LIN {X 0,Y 532.059,Z 786.23,A -85,B 0,C 180,E1 -4333.229,E2 -4333.229} C_VEL
LIN {X 0,Y 530.415,Z 776.665,A -85,B 0,C 180,E1 -4333.53,E2 -4333.53} C_VEL
LIN {X 0,Y 530.416,Z 773.451,A -85,B 0,C 180,E1 -4336.156,E2 -4336.156} C_VEL
LIN {X 0,Y 530.403,Z 770.567,A -85,B 0,C 180,E1 -4338.543,E2 -4338.543} C_VEL
LIN {X 0,Y 530.453,Z 767.793,A -85,B 0,C 180,E1 -4340.961,E2 -4340.961} C_VEL
LIN {X 0,Y 530.507,Z 764.565,A -85,B 0,C 180,E1 -4343.922,E2 -4343.922} C_VEL
LIN {X 0,Y 530.506,Z 761.259,A -85,B 0,C 180,E1 -4346.771,E2 -4346.771} C_VEL
LIN {X 0,Y 530.49,Z 757.968,A -85,B 0,C 180,E1 -4349.353,E2 -4349.353} C_VEL
LIN {X 0,Y 530.48,Z 755.565,A -85,B 0,C 180,E1 -4351.111,E2 -4351.111} C_VEL
LIN {X 0,Y 530.791,Z 755.371,A -85,B 0,C 180,E1 -4353.788,E2 -4353.788} C_VEL
LIN {X 0,Y 530.947,Z 755.346,A -85,B 0,C 180,E1 -4356.56,E2 -4356.56} C_VEL
LIN {X 0,Y 530.992,Z 755.343,A -85,B 0,C 180,E1 -4359.444,E2 -4359.444} C_VEL
LIN {X 0,Y 530.968,Z 755.343,A -85,B 0,C 180,E1 -4362.458,E2 -4362.458} C_VEL
LIN {X 0,Y 530.99,Z 755.342,A -85,B 0,C 180,E1 -4365.453,E2 -4365.453} C_VEL
LIN {X 0,Y 530.998,Z 755.342,A -85,B 0,C 180,E1 -4368.565,E2 -4368.565} C_VEL
LIN {X 0,Y 530.992,Z 755.408,A -85,B 0,C 180,E1 -4371.744,E2 -4371.744} C_VEL
LIN {X 0,Y 532.042,Z 761.565,A -85,B 0,C 180,E1 -4374.093,E2 -4374.093} C_VEL
LIN {X 0,Y 532.013,Z 767.898,A -85,B 0,C 180,E1 -4376.33,E2 -4376.33} C_VEL
LIN {X 0,Y 531.734,Z 776.441,A -85,B 0,C 180,E1 -4379.218,E2 -4379.218} C_VEL
LIN {X 0,Y 531.516,Z 785.016,A -85,B 0,C 180,E1 -4382.005,E2 -4382.005} C_VEL
LIN {X 0,Y 531.294,Z 794.397,A -85,B 0,C 180,E1 -4384.957,E2 -4384.957} C_VEL
LIN {X 0,Y 531.163,Z 803.886,A -85,B 0,C 180,E1 -4387.85,E2 -4387.85} C_VEL
LIN {X 0,Y 530.969,Z 813.168,A -85,B 0,C 180,E1 -4390.676,E2 -4390.676} C_VEL
LIN {X 0,Y 530.828,Z 822.435,A -85,B 0,C 180,E1 -4393.462,E2 -4393.462} C_VEL
LIN {X 0,Y 530.706,Z 832.53,A -85,B 0,C 180,E1 -4396.454,E2 -4396.454} C_VEL
LIN {X 0,Y 532.33,Z 843.349,A -85,B 0,C 180,E1 -4396.739,E2 -4396.739} C_VEL
LIN {X 0,Y 532.127,Z 856.77,A -85,B 0,C 180,E1 -4397.171,E2 -4397.171} C_VEL
LIN {X 0,Y 531.869,Z 868.408,A -85,B 0,C 180,E1 -4397.697,E2 -4397.697} C_VEL
LIN {X 0,Y 531.655,Z 879.403,A -85,B 0,C 180,E1 -4398.347,E2 -4398.347} C_VEL
LIN {X 0,Y 531.411,Z 890.095,A -85,B 0,C 180,E1 -4399.137,E2 -4399.137} C_VEL
LIN {X 0,Y 531.128,Z 900.539,A -85,B 0,C 180,E1 -4400.095,E2 -4400.095} C_VEL
LIN {X 0,Y 530.931,Z 908.991,A -85,B 0,C 180,E1 -4401.052,E2 -4401.052} C_VEL
LIN {X 0,Y 530.759,Z 917.236,A -85,B 0,C 180,E1 -4402.199,E2 -4402.199} C_VEL
LIN {X 0,Y 530.599,Z 924.271,A -85,B 0,C 180,E1 -4403.42,E2 -4403.42} C_VEL
LIN {X 0,Y 530.525,Z 929.95,A -85,B 0,C 180,E1 -4404.679,E2 -4404.679} C_VEL
LIN {X 0,Y 530.523,Z 933.895,A -85,B 0,C 180,E1 -4405.822,E2 -4405.822} C_VEL
LIN {X 0,Y 530.457,Z 936.807,A -85,B 0,C 180,E1 -4406.962,E2 -4406.962} C_VEL
LIN {X 0,Y 530.41,Z 938.196,A -85,B 0,C 180,E1 -4407.722,E2 -4407.722} C_VEL
LIN {X 0,Y 530.344,Z 939.786,A -85,B 0,C 180,E1 -4409.241,E2 -4409.241} C_VEL
LIN {X 0,Y 530.343,Z 940,A -85,B 0,C 180,E1 -4410,E2 -4410} C_VEL
LIN {X 0,Y 530.361,Z 939.185,A -85,B 0,C 180,E1 -4411.519,E2 -4411.519} C_VEL
LIN {X 0,Y 530.41,Z 938.198,A -85,B 0,C 180,E1 -4412.278,E2 -4412.278} C_VEL
LIN {X 0,Y 530.457,Z 936.81,A -85,B 0,C 180,E1 -4413.038,E2 -4413.038} C_VEL
LIN {X 0,Y 530.523,Z 933.895,A -85,B 0,C 180,E1 -4414.178,E2 -4414.178} C_VEL
LIN {X 0,Y 530.525,Z 929.948,A -85,B 0,C 180,E1 -4415.321,E2 -4415.321} C_VEL
LIN {X 0,Y 530.599,Z 924.268,A -85,B 0,C 180,E1 -4416.581,E2 -4416.581} C_VEL
LIN {X 0,Y 530.759,Z 917.236,A -85,B 0,C 180,E1 -4417.801,E2 -4417.801} C_VEL
LIN {X 0,Y 530.931,Z 908.991,A -85,B 0,C 180,E1 -4418.948,E2 -4418.948} C_VEL
LIN {X 0,Y 531.112,Z 900.539,A -85,B 0,C 180,E1 -4419.906,E2 -4419.906} C_VEL
LIN {X 0,Y 531.411,Z 890.094,A -85,B 0,C 180,E1 -4420.863,E2 -4420.863} C_VEL
LIN {X 0,Y 531.696,Z 878.247,A -85,B 0,C 180,E1 -4421.731,E2 -4421.731} C_VEL
LIN {X 0,Y 531.921,Z 866.488,A -85,B 0,C 180,E1 -4422.398,E2 -4422.398} C_VEL
LIN {X 0,Y 532.161,Z 854.165,A -85,B 0,C 180,E1 -4422.926,E2 -4422.926} C_VEL
LIN {X 0,Y 532.183,Z 841.514,A -85,B 0,C 180,E1 -4423.314,E2 -4423.314} C_VEL
LIN {X 0,Y 530.706,Z 832.53,A -85,B 0,C 180,E1 -4423.546,E2 -4423.546} C_VEL
LIN {X 0,Y 530.828,Z 822.435,A -85,B 0,C 180,E1 -4426.538,E2 -4426.538} C_VEL
LIN {X 0,Y 530.968,Z 813.168,A -85,B 0,C 180,E1 -4429.324,E2 -4429.324} C_VEL
LIN {X 0,Y 531.163,Z 803.882,A -85,B 0,C 180,E1 -4432.15,E2 -4432.15} C_VEL
LIN {X 0,Y 531.268,Z 794.03,A -85,B 0,C 180,E1 -4435.044,E2 -4435.044} C_VEL
LIN {X 0,Y 531.414,Z 784.276,A -85,B 0,C 180,E1 -4438.001,E2 -4438.001} C_VEL
LIN {X 0,Y 531.62,Z 774.782,A -85,B 0,C 180,E1 -4441.036,E2 -4441.036} C_VEL
LIN {X 0,Y 531.858,Z 767.114,A -85,B 0,C 180,E1 -4443.71,E2 -4443.71} C_VEL
LIN {X 0,Y 532.032,Z 762.369,A -85,B 0,C 180,E1 -4445.537,E2 -4445.537} C_VEL
LIN {X 0,Y 531.466,Z 758.043,A -85,B 0,C 180,E1 -4447.492,E2 -4447.492} C_VEL
LIN {X 0,Y 530.983,Z 755.347,A -85,B 0,C 180,E1 -4449.015,E2 -4449.015} C_VEL
LIN {X 0,Y 530.987,Z 755.344,A -85,B 0,C 180,E1 -4452.166,E2 -4452.166} C_VEL
LIN {X 0,Y 530.989,Z 755.345,A -85,B 0,C 180,E1 -4455.453,E2 -4455.453} C_VEL
LIN {X 0,Y 530.983,Z 755.345,A -85,B 0,C 180,E1 -4458.563,E2 -4458.563} C_VEL
LIN {X 0,Y 530.959,Z 755.347,A -85,B 0,C 180,E1 -4461.529,E2 -4461.529} C_VEL
LIN {X 0,Y 530.929,Z 755.353,A -85,B 0,C 180,E1 -4464.377,E2 -4464.377} C_VEL
LIN {X 0,Y 530.909,Z 755.357,A -85,B 0,C 180,E1 -4465.304,E2 -4465.304} C_VEL
LIN {X 0,Y 530.826,Z 756.592,A -85,B 0,C 180,E1 -4467.123,E2 -4467.123} C_VEL
LIN {X 0,Y 530.714,Z 759.006,A -85,B 0,C 180,E1 -4469.786,E2 -4469.786} C_VEL
LIN {X 0,Y 530.622,Z 761.58,A -85,B 0,C 180,E1 -4472.549,E2 -4472.549} C_VEL
LIN {X 0,Y 530.564,Z 763.83,A -85,B 0,C 180,E1 -4474.92,E2 -4474.92} C_VEL
LIN {X 0,Y 530.51,Z 766.833,A -85,B 0,C 180,E1 -4478.024,E2 -4478.024} C_VEL
LIN {X 0,Y 530.425,Z 769.498,A -85,B 0,C 180,E1 -4480.655,E2 -4480.655} C_VEL
LIN {X 0,Y 530.429,Z 772.38,A -85,B 0,C 180,E1 -4483.052,E2 -4483.052} C_VEL
LIN {X 0,Y 530.43,Z 776.224,A -85,B 0,C 180,E1 -4486.202,E2 -4486.202} C_VEL
LIN {X 0,Y 530.44,Z 776.674,A -85,B 0,C 180,E1 -4486.568,E2 -4486.568} C_VEL
LIN {X 0,Y 532.261,Z 788.537,A -85,B 0,C 180,E1 -4486.931,E2 -4486.931} C_VEL
LIN {X 0,Y 532.013,Z 801.428,A -85,B 0,C 180,E1 -4487.41,E2 -4487.41} C_VEL
LIN {X 0,Y 531.83,Z 813.17,A -85,B 0,C 180,E1 -4488.005,E2 -4488.005} C_VEL
LIN {X 0,Y 531.551,Z 824.586,A -85,B 0,C 180,E1 -4488.753,E2 -4488.753} C_VEL
LIN {X 0,Y 531.282,Z 835.099,A -85,B 0,C 180,E1 -4489.616,E2 -4489.616} C_VEL
LIN {X 0,Y 531.071,Z 843.691,A -85,B 0,C 180,E1 -4490.478,E2 -4490.478} C_VEL
LIN {X 0,Y 530.892,Z 851.608,A -85,B 0,C 180,E1 -4491.434,E2 -4491.434} C_VEL
LIN {X 0,Y 530.69,Z 859.354,A -85,B 0,C 180,E1 -4492.58,E2 -4492.58} C_VEL
LIN {X 0,Y 530.603,Z 866.462,A -85,B 0,C 180,E1 -4493.917,E2 -4493.917} C_VEL
LIN {X 0,Y 530.46,Z 871.201,A -85,B 0,C 180,E1 -4495.059,E2 -4495.059} C_VEL
LIN {X 0,Y 530.516,Z 874.833,A -85,B 0,C 180,E1 -4496.201,E2 -4496.201} C_VEL
LIN {X 0,Y 530.458,Z 876.708,A -85,B 0,C 180,E1 -4496.961,E2 -4496.961} C_VEL
LIN {X 0,Y 530.411,Z 878.13,A -85,B 0,C 180,E1 -4497.721,E2 -4497.721} C_VEL
LIN {X 0,Y 530.345,Z 879.758,A -85,B 0,C 180,E1 -4499.24,E2 -4499.24} C_VEL
LIN {X 0,Y 530.343,Z 879.996,A -85,B 0,C 180,E1 -4499.999,E2 -4499.999} C_VEL
LIN {X 0,Y 530.344,Z 879.814,A -85,B 0,C 180,E1 -4500.759,E2 -4500.759} C_VEL
LIN {X 0,Y 530.41,Z 878.263,A -85,B 0,C 180,E1 -4502.277,E2 -4502.277} C_VEL
LIN {X 0,Y 530.457,Z 876.902,A -85,B 0,C 180,E1 -4503.037,E2 -4503.037} C_VEL
LIN {X 0,Y 530.523,Z 874.023,A -85,B 0,C 180,E1 -4504.177,E2 -4504.177} C_VEL
LIN {X 0,Y 530.523,Z 870.121,A -85,B 0,C 180,E1 -4505.32,E2 -4505.32} C_VEL
LIN {X 0,Y 530.592,Z 864.537,A -85,B 0,C 180,E1 -4506.575,E2 -4506.575} C_VEL
LIN {X 0,Y 530.757,Z 857.531,A -85,B 0,C 180,E1 -4507.8,E2 -4507.8} C_VEL
LIN {X 0,Y 530.927,Z 849.347,A -85,B 0,C 180,E1 -4508.947,E2 -4508.947} C_VEL
LIN {X 0,Y 531.106,Z 840.977,A -85,B 0,C 180,E1 -4509.905,E2 -4509.905} C_VEL
LIN {X 0,Y 531.404,Z 830.653,A -85,B 0,C 180,E1 -4510.862,E2 -4510.862} C_VEL
LIN {X 0,Y 531.643,Z 818.958,A -85,B 0,C 180,E1 -4511.729,E2 -4511.729} C_VEL
LIN {X 0,Y 531.868,Z 807.425,A -85,B 0,C 180,E1 -4512.398,E2 -4512.398} C_VEL
LIN {X 0,Y 532.131,Z 795.405,A -85,B 0,C 180,E1 -4512.925,E2 -4512.925} C_VEL
LIN {X 0,Y 532.125,Z 786.435,A -85,B 0,C 180,E1 -4513.229,E2 -4513.229} C_VEL
LIN {X 0,Y 530.414,Z 776.667,A -85,B 0,C 180,E1 -4513.529,E2 -4513.529} C_VEL
LIN {X 0,Y 530.411,Z 773.452,A -85,B 0,C 180,E1 -4516.155,E2 -4516.155} C_VEL
LIN {X 0,Y 530.399,Z 770.569,A -85,B 0,C 180,E1 -4518.542,E2 -4518.542} C_VEL
LIN {X 0,Y 530.441,Z 767.695,A -85,B 0,C 180,E1 -4520.96,E2 -4520.96} C_VEL
LIN {X 0,Y 530.514,Z 764.314,A -85,B 0,C 180,E1 -4523.924,E2 -4523.924} C_VEL
LIN {X 0,Y 530.526,Z 761.426,A -85,B 0,C 180,E1 -4526.769,E2 -4526.769} C_VEL
LIN {X 0,Y 530.558,Z 758.697,A -85,B 0,C 180,E1 -4529.347,E2 -4529.347} C_VEL
LIN {X 0,Y 530.622,Z 755.781,A -85,B 0,C 180,E1 -4532.04,E2 -4532.04} C_VEL
LIN {X 0,Y 530.783,Z 755.372,A -85,B 0,C 180,E1 -4533.786,E2 -4533.786} C_VEL
LIN {X 0,Y 530.941,Z 755.345,A -85,B 0,C 180,E1 -4536.558,E2 -4536.558} C_VEL
LIN {X 0,Y 530.975,Z 755.344,A -85,B 0,C 180,E1 -4539.57,E2 -4539.57} C_VEL
LIN {X 0,Y 530.3,Z 755.427,A -85,B 0,C 180,E1 -4540.203,E2 -4540.203} C_VEL
LIN {X 0,Y 527.438,Z 755.788,A -85,B 0,C 180,E1 -4541.23,E2 -4541.23} C_VEL
LIN {X 0,Y 525.026,Z 756.084,A -85,B 0,C 180,E1 -4542.057,E2 -4542.057} C_VEL
LIN {X 0,Y 523.992,Z 756.212,A -85,B 0,C 180,E1 -4542.696,E2 -4542.696} C_VEL
LIN {X 0,Y 523.909,Z 756.224,A -85,B 0,C 180,E1 -4542.912,E2 -4542.912} C_VEL
LIN {X 0,Y 523.936,Z 756.221,A -85,B 0,C 180,E1 -4545.771,E2 -4545.771} C_VEL
LIN {X 0,Y 523.932,Z 756.22,A -85,B 0,C 180,E1 -4548.907,E2 -4548.907} C_VEL
LIN {X 0,Y 523.908,Z 756.223,A -85,B 0,C 180,E1 -4551.897,E2 -4551.897} C_VEL
LIN {X 0,Y 523.916,Z 756.221,A -85,B 0,C 180,E1 -4554.911,E2 -4554.911} C_VEL
LIN {X 0,Y 523.927,Z 756.224,A -85,B 0,C 180,E1 -4557.679,E2 -4557.679} C_VEL
LIN {X 0,Y 523.945,Z 756.216,A -85,B 0,C 180,E1 -4560.676,E2 -4560.676} C_VEL
LIN {X 0,Y 523.925,Z 756.225,A -85,B 0,C 180,E1 -4563.726,E2 -4563.726} C_VEL
LIN {X 0,Y 523.9,Z 756.223,A -85,B 0,C 180,E1 -4566.269,E2 -4566.269} C_VEL
LIN {X 0,Y 523.936,Z 756.216,A -85,B 0,C 180,E1 -4568.766,E2 -4568.766} C_VEL
LIN {X 0,Y 523.928,Z 756.219,A -85,B 0,C 180,E1 -4571.22,E2 -4571.22} C_VEL
LIN {X 0,Y 523.916,Z 756.226,A -85,B 0,C 180,E1 -4573.638,E2 -4573.638} C_VEL
LIN {X 0,Y 523.921,Z 756.224,A -85,B 0,C 180,E1 -4576.027,E2 -4576.027} C_VEL
LIN {X 0,Y 523.979,Z 756.211,A -85,B 0,C 180,E1 -4579.177,E2 -4579.177} C_VEL
LIN {X 0,Y 523.942,Z 756.219,A -85,B 0,C 180,E1 -4581.515,E2 -4581.515} C_VEL
LIN {X 0,Y 524.02,Z 756.206,A -85,B 0,C 180,E1 -4584.613,E2 -4584.613} C_VEL
LIN {X 0,Y 524.093,Z 756.201,A -85,B 0,C 180,E1 -4587.694,E2 -4587.694} C_VEL
LIN {X 0,Y 524.085,Z 756.206,A -85,B 0,C 180,E1 -4590,E2 -4590} C_VEL
LIN {X 0,Y 524.09,Z 756.202,A -85,B 0,C 180,E1 -4592.306,E2 -4592.306} C_VEL
LIN {X 0,Y 523.991,Z 756.218,A -85,B 0,C 180,E1 -4596.16,E2 -4596.16} C_VEL
LIN {X 0,Y 523.933,Z 756.216,A -85,B 0,C 180,E1 -4599.263,E2 -4599.263} C_VEL
LIN {X 0,Y 523.941,Z 756.222,A -85,B 0,C 180,E1 -4602.393,E2 -4602.393} C_VEL
LIN {X 0,Y 523.914,Z 756.219,A -85,B 0,C 180,E1 -4605.563,E2 -4605.563} C_VEL
LIN {X 0,Y 523.906,Z 756.224,A -85,B 0,C 180,E1 -4607.971,E2 -4607.971} C_VEL
LIN {X 0,Y 523.962,Z 756.222,A -85,B 0,C 180,E1 -4610.411,E2 -4610.411} C_VEL
LIN {X 0,Y 523.899,Z 756.223,A -85,B 0,C 180,E1 -4612.894,E2 -4612.894} C_VEL
LIN {X 0,Y 523.89,Z 756.222,A -85,B 0,C 180,E1 -4615.422,E2 -4615.422} C_VEL
LIN {X 0,Y 523.906,Z 756.223,A -85,B 0,C 180,E1 -4618.003,E2 -4618.003} C_VEL
LIN {X 0,Y 523.931,Z 756.222,A -85,B 0,C 180,E1 -4620.854,E2 -4620.854} C_VEL
LIN {X 0,Y 523.922,Z 756.219,A -85,B 0,C 180,E1 -4623.73,E2 -4623.73} C_VEL
LIN {X 0,Y 523.896,Z 756.227,A -85,B 0,C 180,E1 -4626.402,E2 -4626.402} C_VEL
LIN {X 0,Y 523.913,Z 756.223,A -85,B 0,C 180,E1 -4629.086,E2 -4629.086} C_VEL
LIN {X 0,Y 523.945,Z 756.217,A -85,B 0,C 180,E1 -4632.12,E2 -4632.12} C_VEL
LIN {X 0,Y 523.937,Z 756.219,A -85,B 0,C 180,E1 -4635.311,E2 -4635.311} C_VEL
LIN {X 0,Y 523.951,Z 756.221,A -85,B 0,C 180,E1 -4638.691,E2 -4638.691} C_VEL
LIN {X 0,Y 523.912,Z 756.226,A -85,B 0,C 180,E1 -4641.082,E2 -4641.082} C_VEL
LIN {X 0,Y 523.893,Z 756.222,A -85,B 0,C 180,E1 -4643.826,E2 -4643.826} C_VEL
LIN {X 0,Y 523.722,Z 756.251,A -85,B 0,C 180,E1 -4646.621,E2 -4646.621} C_VEL
LIN {X 0,Y 523.505,Z 756.279,A -85,B 0,C 180,E1 -4648.429,E2 -4648.429} C_VEL
LIN {X 0,Y 523.434,Z 759.216,A -85,B 0,C 180,E1 -4651.096,E2 -4651.096} C_VEL
LIN {X 0,Y 523.464,Z 762.594,A -85,B 0,C 180,E1 -4654.098,E2 -4654.098} C_VEL
LIN {X 0,Y 523.385,Z 765.959,A -85,B 0,C 180,E1 -4657.083,E2 -4657.083} C_VEL
LIN {X 0,Y 523.379,Z 769.308,A -85,B 0,C 180,E1 -4660.047,E2 -4660.047} C_VEL
LIN {X 0,Y 523.338,Z 772.383,A -85,B 0,C 180,E1 -4662.817,E2 -4662.817} C_VEL
LIN {X 0,Y 523.364,Z 776.587,A -85,B 0,C 180,E1 -4666.31,E2 -4666.31} C_VEL
LIN {X 0,Y 523.363,Z 776.677,A -85,B 0,C 180,E1 -4666.385,E2 -4666.385} C_VEL
LIN {X 0,Y 525.294,Z 788.698,A -85,B 0,C 180,E1 -4666.756,E2 -4666.756} C_VEL
LIN {X 0,Y 525.059,Z 801.414,A -85,B 0,C 180,E1 -4667.242,E2 -4667.242} C_VEL
LIN {X 0,Y 524.826,Z 811.363,A -85,B 0,C 180,E1 -4667.742,E2 -4667.742} C_VEL
LIN {X 0,Y 524.67,Z 821.852,A -85,B 0,C 180,E1 -4668.41,E2 -4668.41} C_VEL
LIN {X 0,Y 524.401,Z 830.657,A -85,B 0,C 180,E1 -4669.089,E2 -4669.089} C_VEL
LIN {X 0,Y 524.179,Z 838.123,A -85,B 0,C 180,E1 -4669.768,E2 -4669.768} C_VEL
LIN {X 0,Y 523.99,Z 845.395,A -85,B 0,C 180,E1 -4670.544,E2 -4670.544} C_VEL
LIN {X 0,Y 523.794,Z 852.985,A -85,B 0,C 180,E1 -4671.513,E2 -4671.513} C_VEL
LIN {X 0,Y 523.636,Z 859.318,A -85,B 0,C 180,E1 -4672.482,E2 -4672.482} C_VEL
LIN {X 0,Y 523.528,Z 864.446,A -85,B 0,C 180,E1 -4673.415,E2 -4673.415} C_VEL
LIN {X 0,Y 523.464,Z 869.72,A -85,B 0,C 180,E1 -4674.608,E2 -4674.608} C_VEL
LIN {X 0,Y 523.441,Z 873.701,A -85,B 0,C 180,E1 -4675.766,E2 -4675.766} C_VEL
LIN {X 0,Y 523.367,Z 876.652,A -85,B 0,C 180,E1 -4676.922,E2 -4676.922} C_VEL
LIN {X 0,Y 523.334,Z 878.143,A -85,B 0,C 180,E1 -4677.692,E2 -4677.692} C_VEL
LIN {X 0,Y 523.25,Z 879.719,A -85,B 0,C 180,E1 -4679.231,E2 -4679.231} C_VEL
LIN {X 0,Y 523.247,Z 879.999,A -85,B 0,C 180,E1 -4680.001,E2 -4680.001} C_VEL
LIN {X 0,Y 523.275,Z 879.2,A -85,B 0,C 180,E1 -4681.54,E2 -4681.54} C_VEL
LIN {X 0,Y 523.334,Z 878.278,A -85,B 0,C 180,E1 -4682.31,E2 -4682.31} C_VEL
LIN {X 0,Y 523.444,Z 875.036,A -85,B 0,C 180,E1 -4683.85,E2 -4683.85} C_VEL
LIN {X 0,Y 523.383,Z 871.477,A -85,B 0,C 180,E1 -4685.008,E2 -4685.008} C_VEL
LIN {X 0,Y 523.537,Z 868.573,A -85,B 0,C 180,E1 -4685.779,E2 -4685.779} C_VEL
LIN {X 0,Y 523.584,Z 862.019,A -85,B 0,C 180,E1 -4687.133,E2 -4687.133} C_VEL
LIN {X 0,Y 523.723,Z 856.229,A -85,B 0,C 180,E1 -4688.101,E2 -4688.101} C_VEL
LIN {X 0,Y 523.867,Z 849.264,A -85,B 0,C 180,E1 -4689.07,E2 -4689.07} C_VEL
LIN {X 0,Y 524.051,Z 842.707,A -85,B 0,C 180,E1 -4689.846,E2 -4689.846} C_VEL
LIN {X 0,Y 524.285,Z 833.886,A -85,B 0,C 180,E1 -4690.72,E2 -4690.72} C_VEL
LIN {X 0,Y 524.545,Z 825.715,A -85,B 0,C 180,E1 -4691.399,E2 -4691.399} C_VEL
LIN {X 0,Y 524.715,Z 816.442,A -85,B 0,C 180,E1 -4692.043,E2 -4692.043} C_VEL
LIN {X 0,Y 524.97,Z 807.257,A -85,B 0,C 180,E1 -4692.566,E2 -4692.566} C_VEL
LIN {X 0,Y 525.192,Z 796.453,A -85,B 0,C 180,E1 -4693.052,E2 -4693.052} C_VEL
LIN {X 0,Y 525.151,Z 787.293,A -85,B 0,C 180,E1 -4693.376,E2 -4693.376} C_VEL
LIN {X 0,Y 523.353,Z 776.664,A -85,B 0,C 180,E1 -4693.716,E2 -4693.716} C_VEL
LIN {X 0,Y 523.315,Z 773.45,A -85,B 0,C 180,E1 -4696.382,E2 -4696.382} C_VEL
LIN {X 0,Y 523.315,Z 770.726,A -85,B 0,C 180,E1 -4698.804,E2 -4698.804} C_VEL
LIN {X 0,Y 523.384,Z 768.119,A -85,B 0,C 180,E1 -4701.258,E2 -4701.258} C_VEL
LIN {X 0,Y 523.429,Z 765.314,A -85,B 0,C 180,E1 -4703.754,E2 -4703.754} C_VEL
LIN {X 0,Y 523.431,Z 762.363,A -85,B 0,C 180,E1 -4706.301,E2 -4706.301} C_VEL
LIN {X 0,Y 523.417,Z 758.654,A -85,B 0,C 180,E1 -4709.218,E2 -4709.218} C_VEL
LIN {X 0,Y 523.396,Z 756.574,A -85,B 0,C 180,E1 -4710.753,E2 -4710.753} C_VEL
LIN {X 0,Y 523.597,Z 756.267,A -85,B 0,C 180,E1 -4712.474,E2 -4712.474} C_VEL
LIN {X 0,Y 523.865,Z 756.234,A -85,B 0,C 180,E1 -4715.232,E2 -4715.232} C_VEL
LIN {X 0,Y 523.919,Z 756.22,A -85,B 0,C 180,E1 -4718.102,E2 -4718.102} C_VEL
LIN {X 0,Y 523.939,Z 756.224,A -85,B 0,C 180,E1 -4721.093,E2 -4721.093} C_VEL
LIN {X 0,Y 523.939,Z 756.218,A -85,B 0,C 180,E1 -4724.229,E2 -4724.229} C_VEL
LIN {X 0,Y 523.922,Z 756.226,A -85,B 0,C 180,E1 -4726.833,E2 -4726.833} C_VEL
LIN {X 0,Y 523.944,Z 756.224,A -85,B 0,C 180,E1 -4728.908,E2 -4728.908} C_VEL
LIN {X 0,Y 523.949,Z 756.275,A -85,B 0,C 180,E1 -4731.472,E2 -4731.472} C_VEL
LIN {X 0,Y 525.035,Z 762.583,A -85,B 0,C 180,E1 -4733.916,E2 -4733.916} C_VEL
LIN {X 0,Y 525.09,Z 767.758,A -85,B 0,C 180,E1 -4735.796,E2 -4735.796} C_VEL
LIN {X 0,Y 524.805,Z 775.632,A -85,B 0,C 180,E1 -4738.515,E2 -4738.515} C_VEL
LIN {X 0,Y 524.524,Z 784.894,A -85,B 0,C 180,E1 -4741.598,E2 -4741.598} C_VEL
LIN {X 0,Y 524.328,Z 793.131,A -85,B 0,C 180,E1 -4744.249,E2 -4744.249} C_VEL
LIN {X 0,Y 524.129,Z 802.291,A -85,B 0,C 180,E1 -4747.116,E2 -4747.116} C_VEL
LIN {X 0,Y 523.996,Z 811.37,A -85,B 0,C 180,E1 -4749.862,E2 -4749.862} C_VEL
LIN {X 0,Y 523.821,Z 821.111,A -85,B 0,C 180,E1 -4752.832,E2 -4752.832} C_VEL
LIN {X 0,Y 523.659,Z 831.703,A -85,B 0,C 180,E1 -4756.02,E2 -4756.02} C_VEL
LIN {X 0,Y 523.652,Z 832.725,A -85,B 0,C 180,E1 -4756.286,E2 -4756.286} C_VEL
LIN {X 0,Y 525.427,Z 844.264,A -85,B 0,C 180,E1 -4756.586,E2 -4756.586} C_VEL
LIN {X 0,Y 525.216,Z 856.771,A -85,B 0,C 180,E1 -4756.999,E2 -4756.999} C_VEL
LIN {X 0,Y 524.934,Z 868.407,A -85,B 0,C 180,E1 -4757.532,E2 -4757.532} C_VEL
LIN {X 0,Y 524.684,Z 879.822,A -85,B 0,C 180,E1 -4758.218,E2 -4758.218} C_VEL
LIN {X 0,Y 524.395,Z 891.264,A -85,B 0,C 180,E1 -4759.088,E2 -4759.088} C_VEL
LIN {X 0,Y 524.106,Z 900.539,A -85,B 0,C 180,E1 -4759.961,E2 -4759.961} C_VEL
LIN {X 0,Y 523.897,Z 908.991,A -85,B 0,C 180,E1 -4760.931,E2 -4760.931} C_VEL
LIN {X 0,Y 523.689,Z 917.236,A -85,B 0,C 180,E1 -4762.093,E2 -4762.093} C_VEL
LIN {X 0,Y 523.576,Z 922.868,A -85,B 0,C 180,E1 -4763.061,E2 -4763.061} C_VEL
LIN {X 0,Y 523.544,Z 928.366,A -85,B 0,C 180,E1 -4764.222,E2 -4764.222} C_VEL
LIN {X 0,Y 523.361,Z 932.677,A -85,B 0,C 180,E1 -4765.379,E2 -4765.379} C_VEL
LIN {X 0,Y 523.444,Z 934.958,A -85,B 0,C 180,E1 -4766.151,E2 -4766.151} C_VEL
LIN {X 0,Y 523.368,Z 936.807,A -85,B 0,C 180,E1 -4766.921,E2 -4766.921} C_VEL
LIN {X 0,Y 523.334,Z 938.195,A -85,B 0,C 180,E1 -4767.691,E2 -4767.691} C_VEL
LIN {X 0,Y 523.25,Z 939.786,A -85,B 0,C 180,E1 -4769.23,E2 -4769.23} C_VEL
LIN {X 0,Y 523.246,Z 940,A -85,B 0,C 180,E1 -4770,E2 -4770} C_VEL
LIN {X 0,Y 523.275,Z 939.185,A -85,B 0,C 180,E1 -4771.539,E2 -4771.539} C_VEL
LIN {X 0,Y 523.334,Z 938.197,A -85,B 0,C 180,E1 -4772.309,E2 -4772.309} C_VEL
LIN {X 0,Y 523.368,Z 936.81,A -85,B 0,C 180,E1 -4773.079,E2 -4773.079} C_VEL
LIN {X 0,Y 523.442,Z 933.895,A -85,B 0,C 180,E1 -4774.235,E2 -4774.235} C_VEL
LIN {X 0,Y 523.464,Z 929.948,A -85,B 0,C 180,E1 -4775.393,E2 -4775.393} C_VEL
LIN {X 0,Y 523.524,Z 924.731,A -85,B 0,C 180,E1 -4776.58,E2 -4776.58} C_VEL
LIN {X 0,Y 523.666,Z 918.467,A -85,B 0,C 180,E1 -4777.713,E2 -4777.713} C_VEL
LIN {X 0,Y 523.857,Z 910.477,A -85,B 0,C 180,E1 -4778.875,E2 -4778.875} C_VEL
LIN {X 0,Y 524.085,Z 902.333,A -85,B 0,C 180,E1 -4779.845,E2 -4779.845} C_VEL
LIN {X 0,Y 524.365,Z 892.398,A -85,B 0,C 180,E1 -4780.815,E2 -4780.815} C_VEL
LIN {X 0,Y 524.666,Z 881.218,A -85,B 0,C 180,E1 -4781.686,E2 -4781.686} C_VEL
LIN {X 0,Y 524.901,Z 870.172,A -85,B 0,C 180,E1 -4782.37,E2 -4782.37} C_VEL
LIN {X 0,Y 525.171,Z 857.973,A -85,B 0,C 180,E1 -4782.953,E2 -4782.953} C_VEL
LIN {X 0,Y 525.387,Z 845.172,A -85,B 0,C 180,E1 -4783.391,E2 -4783.391} C_VEL
LIN {X 0,Y 524.969,Z 840.5,A -85,B 0,C 180,E1 -4783.525,E2 -4783.525} C_VEL
LIN {X 0,Y 523.641,Z 832.53,A -85,B 0,C 180,E1 -4783.733,E2 -4783.733} C_VEL
LIN {X 0,Y 523.796,Z 822.435,A -85,B 0,C 180,E1 -4786.767,E2 -4786.767} C_VEL
LIN {X 0,Y 523.96,Z 813.168,A -85,B 0,C 180,E1 -4789.593,E2 -4789.593} C_VEL
LIN {X 0,Y 524.124,Z 803.086,A -85,B 0,C 180,E1 -4792.545,E2 -4792.545} C_VEL
LIN {X 0,Y 524.252,Z 792.491,A -85,B 0,C 180,E1 -4795.745,E2 -4795.745} C_VEL
LIN {X 0,Y 524.394,Z 783.918,A -85,B 0,C 180,E1 -4798.41,E2 -4798.41} C_VEL
LIN {X 0,Y 524.649,Z 774.575,A -85,B 0,C 180,E1 -4801.495,E2 -4801.495} C_VEL
LIN {X 0,Y 524.95,Z 767.089,A -85,B 0,C 180,E1 -4804.215,E2 -4804.215} C_VEL
LIN {X 0,Y 524.989,Z 762.525,A -85,B 0,C 180,E1 -4806.088,E2 -4806.088} C_VEL
LIN {X 0,Y 524.324,Z 758.472,A -85,B 0,C 180,E1 -4808.067,E2 -4808.067} C_VEL
LIN {X 0,Y 523.958,Z 756.222,A -85,B 0,C 180,E1 -4809.454,E2 -4809.454} C_VEL
LIN {X 0,Y 523.94,Z 756.223,A -85,B 0,C 180,E1 -4812.459,E2 -4812.459} C_VEL
LIN {X 0,Y 523.958,Z 756.222,A -85,B 0,C 180,E1 -4815.309,E2 -4815.309} C_VEL
LIN {X 0,Y 523.944,Z 756.224,A -85,B 0,C 180,E1 -4818.692,E2 -4818.692} C_VEL
LIN {X 0,Y 523.918,Z 756.223,A -85,B 0,C 180,E1 -4821.898,E2 -4821.898} C_VEL
LIN {X 0,Y 523.866,Z 756.234,A -85,B 0,C 180,E1 -4824.921,E2 -4824.921} C_VEL
LIN {X 0,Y 523.805,Z 756.314,A -85,B 0,C 180,E1 -4825.7,E2 -4825.7} C_VEL
LIN {X 0,Y 523.715,Z 758.673,A -85,B 0,C 180,E1 -4828.441,E2 -4828.441} C_VEL
LIN {X 0,Y 523.63,Z 761.076,A -85,B 0,C 180,E1 -4831.106,E2 -4831.106} C_VEL
LIN {X 0,Y 523.531,Z 763.833,A -85,B 0,C 180,E1 -4834.083,E2 -4834.083} C_VEL
LIN {X 0,Y 523.449,Z 766.738,A -85,B 0,C 180,E1 -4837.084,E2 -4837.084} C_VEL
LIN {X 0,Y 523.384,Z 769.554,A -85,B 0,C 180,E1 -4840.046,E2 -4840.046} C_VEL
LIN {X 0,Y 523.342,Z 772.381,A -85,B 0,C 180,E1 -4842.815,E2 -4842.815} C_VEL
LIN {X 0,Y 523.341,Z 776.465,A -85,B 0,C 180,E1 -4846.209,E2 -4846.209} C_VEL
LIN {X 0,Y 523.344,Z 776.675,A -85,B 0,C 180,E1 -4846.382,E2 -4846.382} C_VEL
LIN {X 0,Y 525.347,Z 789.317,A -85,B 0,C 180,E1 -4846.78,E2 -4846.78} C_VEL
LIN {X 0,Y 525.09,Z 801.442,A -85,B 0,C 180,E1 -4847.241,E2 -4847.241} C_VEL
LIN {X 0,Y 524.888,Z 812.537,A -85,B 0,C 180,E1 -4847.806,E2 -4847.806} C_VEL
LIN {X 0,Y 524.585,Z 824.593,A -85,B 0,C 180,E1 -4848.602,E2 -4848.602} C_VEL
LIN {X 0,Y 524.284,Z 835.105,A -85,B 0,C 180,E1 -4849.476,E2 -4849.476} C_VEL
LIN {X 0,Y 524.061,Z 843.697,A -85,B 0,C 180,E1 -4850.349,E2 -4850.349} C_VEL
LIN {X 0,Y 523.86,Z 851.613,A -85,B 0,C 180,E1 -4851.319,E2 -4851.319} C_VEL
LIN {X 0,Y 523.637,Z 859.358,A -85,B 0,C 180,E1 -4852.48,E2 -4852.48} C_VEL
LIN {X 0,Y 523.517,Z 866.465,A -85,B 0,C 180,E1 -4853.834,E2 -4853.834} C_VEL
LIN {X 0,Y 523.384,Z 871.203,A -85,B 0,C 180,E1 -4854.992,E2 -4854.992} C_VEL
LIN {X 0,Y 523.444,Z 874.834,A -85,B 0,C 180,E1 -4856.15,E2 -4856.15} C_VEL
LIN {X 0,Y 523.368,Z 876.71,A -85,B 0,C 180,E1 -4856.92,E2 -4856.92} C_VEL
LIN {X 0,Y 523.335,Z 878.13,A -85,B 0,C 180,E1 -4857.69,E2 -4857.69} C_VEL
LIN {X 0,Y 523.251,Z 879.758,A -85,B 0,C 180,E1 -4859.23,E2 -4859.23} C_VEL
LIN {X 0,Y 523.247,Z 879.997,A -85,B 0,C 180,E1 -4859.999,E2 -4859.999} C_VEL
LIN {X 0,Y 523.25,Z 879.814,A -85,B 0,C 180,E1 -4860.769,E2 -4860.769} C_VEL
LIN {X 0,Y 523.334,Z 878.262,A -85,B 0,C 180,E1 -4862.308,E2 -4862.308} C_VEL
LIN {X 0,Y 523.368,Z 876.9,A -85,B 0,C 180,E1 -4863.078,E2 -4863.078} C_VEL
LIN {X 0,Y 523.441,Z 874.021,A -85,B 0,C 180,E1 -4864.234,E2 -4864.234} C_VEL
LIN {X 0,Y 523.462,Z 870.118,A -85,B 0,C 180,E1 -4865.392,E2 -4865.392} C_VEL
LIN {X 0,Y 523.532,Z 864.375,A -85,B 0,C 180,E1 -4866.691,E2 -4866.691} C_VEL
LIN {X 0,Y 523.687,Z 857.526,A -85,B 0,C 180,E1 -4867.906,E2 -4867.906} C_VEL
LIN {X 0,Y 523.897,Z 849.342,A -85,B 0,C 180,E1 -4869.068,E2 -4869.068} C_VEL
LIN {X 0,Y 524.088,Z 840.971,A -85,B 0,C 180,E1 -4870.039,E2 -4870.039} C_VEL
LIN {X 0,Y 524.418,Z 830.644,A -85,B 0,C 180,E1 -4871.009,E2 -4871.009} C_VEL
LIN {X 0,Y 524.693,Z 820.524,A -85,B 0,C 180,E1 -4871.778,E2 -4871.778} C_VEL
LIN {X 0,Y 524.909,Z 809.232,A -85,B 0,C 180,E1 -4872.467,E2 -4872.467} C_VEL
LIN {X 0,Y 525.167,Z 797.907,A -85,B 0,C 180,E1 -4873.001,E2 -4873.001} C_VEL
LIN {X 0,Y 525.148,Z 787.208,A -85,B 0,C 180,E1 -4873.383,E2 -4873.383} C_VEL
LIN {X 0,Y 523.351,Z 776.666,A -85,B 0,C 180,E1 -4873.715,E2 -4873.715} C_VEL
LIN {X 0,Y 523.311,Z 773.452,A -85,B 0,C 180,E1 -4876.38,E2 -4876.38} C_VEL
LIN {X 0,Y 523.337,Z 769.635,A -85,B 0,C 180,E1 -4879.616,E2 -4879.616} C_VEL
LIN {X 0,Y 523.404,Z 766.858,A -85,B 0,C 180,E1 -4882.104,E2 -4882.104} C_VEL
LIN {X 0,Y 523.424,Z 764.306,A -85,B 0,C 180,E1 -4884.596,E2 -4884.596} C_VEL
LIN {X 0,Y 523.475,Z 761.679,A -85,B 0,C 180,E1 -4887.159,E2 -4887.159} C_VEL
LIN {X 0,Y 523.497,Z 758.794,A -85,B 0,C 180,E1 -4889.783,E2 -4889.783} C_VEL
LIN {X 0,Y 523.552,Z 756.273,A -85,B 0,C 180,E1 -4892.253,E2 -4892.253} C_VEL
LIN {X 0,Y 523.855,Z 756.235,A -85,B 0,C 180,E1 -4895.078,E2 -4895.078} C_VEL
LIN {X 0,Y 523.91,Z 756.22,A -85,B 0,C 180,E1 -4898.101,E2 -4898.101} C_VEL
LIN {X 0,Y 523.935,Z 756.224,A -85,B 0,C 180,E1 -4901.091,E2 -4901.091} C_VEL
LIN {X 0,Y 523.909,Z 756.224,A -85,B 0,C 180,E1 -4902.912,E2 -4902.912} C_VEL
LIN {X 0,Y 523.25,Z 756.311,A -85,B 0,C 180,E1 -4903.554,E2 -4903.554} C_VEL
LIN {X 0,Y 520.411,Z 756.664,A -85,B 0,C 180,E1 -4904.597,E2 -4904.597} C_VEL
LIN {X 0,Y 518.001,Z 756.962,A -85,B 0,C 180,E1 -4905.436,E2 -4905.436} C_VEL
LIN {X 0,Y 516.955,Z 757.088,A -85,B 0,C 180,E1 -4906.085,E2 -4906.085} C_VEL
LIN {X 0,Y 516.864,Z 757.098,A -85,B 0,C 180,E1 -4906.304,E2 -4906.304} C_VEL
LIN {X 0,Y 516.876,Z 757.104,A -85,B 0,C 180,E1 -4909.257,E2 -4909.257} C_VEL
LIN {X 0,Y 516.856,Z 757.099,A -85,B 0,C 180,E1 -4912.273,E2 -4912.273} C_VEL
LIN {X 0,Y 516.871,Z 757.101,A -85,B 0,C 180,E1 -4915.174,E2 -4915.174} C_VEL
LIN {X 0,Y 516.865,Z 757.101,A -85,B 0,C 180,E1 -4917.974,E2 -4917.974} C_VEL
LIN {X 0,Y 516.912,Z 757.092,A -85,B 0,C 180,E1 -4920.695,E2 -4920.695} C_VEL
LIN {X 0,Y 516.891,Z 757.1,A -85,B 0,C 180,E1 -4923.813,E2 -4923.813} C_VEL
LIN {X 0,Y 516.849,Z 757.099,A -85,B 0,C 180,E1 -4926.775,E2 -4926.775} C_VEL
LIN {X 0,Y 516.93,Z 757.097,A -85,B 0,C 180,E1 -4929.731,E2 -4929.731} C_VEL
LIN {X 0,Y 516.887,Z 757.095,A -85,B 0,C 180,E1 -4932.595,E2 -4932.595} C_VEL
LIN {X 0,Y 516.932,Z 757.089,A -85,B 0,C 180,E1 -4935.03,E2 -4935.03} C_VEL
LIN {X 0,Y 516.956,Z 757.089,A -85,B 0,C 180,E1 -4938.233,E2 -4938.233} C_VEL
LIN {X 0,Y 516.919,Z 757.092,A -85,B 0,C 180,E1 -4941.399,E2 -4941.399} C_VEL
LIN {X 0,Y 516.971,Z 757.085,A -85,B 0,C 180,E1 -4944.539,E2 -4944.539} C_VEL
LIN {X 0,Y 517.062,Z 757.076,A -85,B 0,C 180,E1 -4947.663,E2 -4947.663} C_VEL
LIN {X 0,Y 517.054,Z 757.082,A -85,B 0,C 180,E1 -4950,E2 -4950} C_VEL
LIN {X 0,Y 517.06,Z 757.078,A -85,B 0,C 180,E1 -4952.337,E2 -4952.337} C_VEL
LIN {X 0,Y 516.958,Z 757.093,A -85,B 0,C 180,E1 -4956.244,E2 -4956.244} C_VEL
LIN {X 0,Y 516.895,Z 757.093,A -85,B 0,C 180,E1 -4959.39,E2 -4959.39} C_VEL
LIN {X 0,Y 516.894,Z 757.098,A -85,B 0,C 180,E1 -4962.565,E2 -4962.565} C_VEL
LIN {X 0,Y 516.935,Z 757.088,A -85,B 0,C 180,E1 -4965.147,E2 -4965.147} C_VEL
LIN {X 0,Y 516.868,Z 757.104,A -85,B 0,C 180,E1 -4968.224,E2 -4968.224} C_VEL
LIN {X 0,Y 516.903,Z 757.097,A -85,B 0,C 180,E1 -4970.702,E2 -4970.702} C_VEL
LIN {X 0,Y 516.875,Z 757.1,A -85,B 0,C 180,E1 -4974.074,E2 -4974.074} C_VEL
LIN {X 0,Y 516.84,Z 757.107,A -85,B 0,C 180,E1 -4976.663,E2 -4976.663} C_VEL
LIN {X 0,Y 516.9,Z 757.093,A -85,B 0,C 180,E1 -4979.524,E2 -4979.524} C_VEL
LIN {X 0,Y 516.886,Z 757.102,A -85,B 0,C 180,E1 -4982.544,E2 -4982.544} C_VEL
LIN {X 0,Y 516.858,Z 757.099,A -85,B 0,C 180,E1 -4985.33,E2 -4985.33} C_VEL
LIN {X 0,Y 516.873,Z 757.098,A -85,B 0,C 180,E1 -4987.944,E2 -4987.944} C_VEL
LIN {X 0,Y 516.876,Z 757.104,A -85,B 0,C 180,E1 -4990.743,E2 -4990.743} C_VEL
LIN {X 0,Y 516.876,Z 757.104,A -85,B 0,C 180,E1 -4992.832,E2 -4992.832} C_VEL
LIN {X 0,Y 516.889,Z 757.1,A -85,B 0,C 180,E1 -4995.008,E2 -4995.008} C_VEL
LIN {X 0,Y 516.908,Z 757.096,A -85,B 0,C 180,E1 -4998.4,E2 -4998.4} C_VEL
LIN {X 0,Y 516.875,Z 757.1,A -85,B 0,C 180,E1 -5001.285,E2 -5001.285} C_VEL
LIN {X 0,Y 516.819,Z 757.105,A -85,B 0,C 180,E1 -5004.217,E2 -5004.217} C_VEL
LIN {X 0,Y 516.638,Z 757.133,A -85,B 0,C 180,E1 -5007.036,E2 -5007.036} C_VEL
LIN {X 0,Y 516.4,Z 757.427,A -85,B 0,C 180,E1 -5009.027,E2 -5009.027} C_VEL
LIN {X 0,Y 516.368,Z 761.319,A -85,B 0,C 180,E1 -5012.436,E2 -5012.436} C_VEL
LIN {X 0,Y 516.329,Z 764.224,A -85,B 0,C 180,E1 -5015.043,E2 -5015.043} C_VEL
LIN {X 0,Y 516.319,Z 767.268,A -85,B 0,C 180,E1 -5017.759,E2 -5017.759} C_VEL
LIN {X 0,Y 516.305,Z 769.925,A -85,B 0,C 180,E1 -5020.106,E2 -5020.106} C_VEL
LIN {X 0,Y 516.229,Z 773.458,A -85,B 0,C 180,E1 -5023.389,E2 -5023.389} C_VEL
LIN {X 0,Y 516.262,Z 776.678,A -85,B 0,C 180,E1 -5026.194,E2 -5026.194} C_VEL
LIN {X 0,Y 518.329,Z 788.72,A -85,B 0,C 180,E1 -5026.574,E2 -5026.574} C_VEL
LIN {X 0,Y 518.149,Z 801.412,A -85,B 0,C 180,E1 -5027.069,E2 -5027.069} C_VEL
LIN {X 0,Y 517.866,Z 811.793,A -85,B 0,C 180,E1 -5027.601,E2 -5027.601} C_VEL
LIN {X 0,Y 517.697,Z 821.849,A -85,B 0,C 180,E1 -5028.251,E2 -5028.251} C_VEL
LIN {X 0,Y 517.424,Z 830.655,A -85,B 0,C 180,E1 -5028.94,E2 -5028.94} C_VEL
LIN {X 0,Y 517.18,Z 838.12,A -85,B 0,C 180,E1 -5029.628,E2 -5029.628} C_VEL
LIN {X 0,Y 516.975,Z 845.392,A -85,B 0,C 180,E1 -5030.415,E2 -5030.415} C_VEL
LIN {X 0,Y 516.762,Z 852.982,A -85,B 0,C 180,E1 -5031.397,E2 -5031.397} C_VEL
LIN {X 0,Y 516.565,Z 859.316,A -85,B 0,C 180,E1 -5032.378,E2 -5032.378} C_VEL
LIN {X 0,Y 516.449,Z 864.882,A -85,B 0,C 180,E1 -5033.419,E2 -5033.419} C_VEL
LIN {X 0,Y 516.405,Z 869.717,A -85,B 0,C 180,E1 -5034.534,E2 -5034.534} C_VEL
LIN {X 0,Y 516.344,Z 873.697,A -85,B 0,C 180,E1 -5035.708,E2 -5035.708} C_VEL
LIN {X 0,Y 516.282,Z 876.647,A -85,B 0,C 180,E1 -5036.879,E2 -5036.879} C_VEL
LIN {X 0,Y 516.261,Z 878.145,A -85,B 0,C 180,E1 -5037.66,E2 -5037.66} C_VEL
LIN {X 0,Y 516.16,Z 879.713,A -85,B 0,C 180,E1 -5039.221,E2 -5039.221} C_VEL
LIN {X 0,Y 516.154,Z 879.999,A -85,B 0,C 180,E1 -5040.001,E2 -5040.001} C_VEL
LIN {X 0,Y 516.192,Z 879.193,A -85,B 0,C 180,E1 -5041.561,E2 -5041.561} C_VEL
LIN {X 0,Y 516.261,Z 878.278,A -85,B 0,C 180,E1 -5042.341,E2 -5042.341} C_VEL
LIN {X 0,Y 516.355,Z 875.029,A -85,B 0,C 180,E1 -5043.903,E2 -5043.903} C_VEL
LIN {X 0,Y 516.313,Z 871.47,A -85,B 0,C 180,E1 -5045.077,E2 -5045.077} C_VEL
LIN {X 0,Y 516.446,Z 868.572,A -85,B 0,C 180,E1 -5045.859,E2 -5045.859} C_VEL
LIN {X 0,Y 516.508,Z 863.098,A -85,B 0,C 180,E1 -5047.035,E2 -5047.035} C_VEL
LIN {X 0,Y 516.681,Z 856.217,A -85,B 0,C 180,E1 -5048.212,E2 -5048.212} C_VEL
LIN {X 0,Y 516.845,Z 849.251,A -85,B 0,C 180,E1 -5049.195,E2 -5049.195} C_VEL
LIN {X 0,Y 517.028,Z 842.692,A -85,B 0,C 180,E1 -5049.981,E2 -5049.981} C_VEL
LIN {X 0,Y 517.314,Z 833.869,A -85,B 0,C 180,E1 -5050.866,E2 -5050.866} C_VEL
LIN {X 0,Y 517.58,Z 825.696,A -85,B 0,C 180,E1 -5051.554,E2 -5051.554} C_VEL
LIN {X 0,Y 517.773,Z 816.008,A -85,B 0,C 180,E1 -5052.232,E2 -5052.232} C_VEL
LIN {X 0,Y 518.026,Z 807.231,A -85,B 0,C 180,E1 -5052.737,E2 -5052.737} C_VEL
LIN {X 0,Y 518.292,Z 796.423,A -85,B 0,C 180,E1 -5053.229,E2 -5053.229} C_VEL
LIN {X 0,Y 518.217,Z 788.247,A -85,B 0,C 180,E1 -5053.53,E2 -5053.53} C_VEL
LIN {X 0,Y 516.248,Z 776.663,A -85,B 0,C 180,E1 -5053.909,E2 -5053.909} C_VEL
LIN {X 0,Y 516.233,Z 773.652,A -85,B 0,C 180,E1 -5056.613,E2 -5056.613} C_VEL
LIN {X 0,Y 516.249,Z 771.132,A -85,B 0,C 180,E1 -5059.071,E2 -5059.071} C_VEL
LIN {X 0,Y 516.324,Z 768.427,A -85,B 0,C 180,E1 -5061.563,E2 -5061.563} C_VEL
LIN {X 0,Y 516.356,Z 765.419,A -85,B 0,C 180,E1 -5064.227,E2 -5064.227} C_VEL
LIN {X 0,Y 516.368,Z 762.487,A -85,B 0,C 180,E1 -5066.689,E2 -5066.689} C_VEL
LIN {X 0,Y 516.339,Z 758.949,A -85,B 0,C 180,E1 -5069.411,E2 -5069.411} C_VEL
LIN {X 0,Y 516.353,Z 757.17,A -85,B 0,C 180,E1 -5070.964,E2 -5070.964} C_VEL
LIN {X 0,Y 516.743,Z 757.12,A -85,B 0,C 180,E1 -5073.938,E2 -5073.938} C_VEL
LIN {X 0,Y 516.853,Z 757.103,A -85,B 0,C 180,E1 -5076.749,E2 -5076.749} C_VEL
LIN {X 0,Y 516.887,Z 757.098,A -85,B 0,C 180,E1 -5079.722,E2 -5079.722} C_VEL
LIN {X 0,Y 516.909,Z 757.094,A -85,B 0,C 180,E1 -5081.776,E2 -5081.776} C_VEL
LIN {X 0,Y 516.928,Z 757.098,A -85,B 0,C 180,E1 -5085.01,E2 -5085.01} C_VEL
LIN {X 0,Y 516.918,Z 757.094,A -85,B 0,C 180,E1 -5088.399,E2 -5088.399} C_VEL
LIN {X 0,Y 516.9,Z 757.208,A -85,B 0,C 180,E1 -5091.226,E2 -5091.226} C_VEL
LIN {X 0,Y 518.055,Z 763.82,A -85,B 0,C 180,E1 -5093.834,E2 -5093.834} C_VEL
LIN {X 0,Y 518.096,Z 769.28,A -85,B 0,C 180,E1 -5095.84,E2 -5095.84} C_VEL
LIN {X 0,Y 517.788,Z 777.639,A -85,B 0,C 180,E1 -5098.772,E2 -5098.772} C_VEL
LIN {X 0,Y 517.499,Z 786.08,A -85,B 0,C 180,E1 -5101.619,E2 -5101.619} C_VEL
LIN {X 0,Y 517.267,Z 795.419,A -85,B 0,C 180,E1 -5104.66,E2 -5104.66} C_VEL
LIN {X 0,Y 517.074,Z 804.813,A -85,B 0,C 180,E1 -5107.631,E2 -5107.631} C_VEL
LIN {X 0,Y 516.877,Z 814.314,A -85,B 0,C 180,E1 -5110.541,E2 -5110.541} C_VEL
LIN {X 0,Y 516.715,Z 823.759,A -85,B 0,C 180,E1 -5113.404,E2 -5113.404} C_VEL
LIN {X 0,Y 516.603,Z 832.725,A -85,B 0,C 180,E1 -5116.095,E2 -5116.095} C_VEL
LIN {X 0,Y 518.521,Z 845.179,A -85,B 0,C 180,E1 -5116.429,E2 -5116.429} C_VEL
LIN {X 0,Y 518.271,Z 857.98,A -85,B 0,C 180,E1 -5116.871,E2 -5116.871} C_VEL
LIN {X 0,Y 517.949,Z 870.171,A -85,B 0,C 180,E1 -5117.461,E2 -5117.461} C_VEL
LIN {X 0,Y 517.686,Z 881.571,A -85,B 0,C 180,E1 -5118.179,E2 -5118.179} C_VEL
LIN {X 0,Y 517.385,Z 892.398,A -85,B 0,C 180,E1 -5119.037,E2 -5119.037} C_VEL
LIN {X 0,Y 517.056,Z 902.333,A -85,B 0,C 180,E1 -5120.02,E2 -5120.02} C_VEL
LIN {X 0,Y 516.814,Z 911.96,A -85,B 0,C 180,E1 -5121.2,E2 -5121.2} C_VEL
LIN {X 0,Y 516.564,Z 919.621,A -85,B 0,C 180,E1 -5122.377,E2 -5122.377} C_VEL
LIN {X 0,Y 516.427,Z 926.679,A -85,B 0,C 180,E1 -5123.75,E2 -5123.75} C_VEL
LIN {X 0,Y 516.314,Z 931.373,A -85,B 0,C 180,E1 -5124.924,E2 -5124.924} C_VEL
LIN {X 0,Y 516.355,Z 934.958,A -85,B 0,C 180,E1 -5126.098,E2 -5126.098} C_VEL
LIN {X 0,Y 516.283,Z 936.807,A -85,B 0,C 180,E1 -5126.879,E2 -5126.879} C_VEL
LIN {X 0,Y 516.261,Z 938.194,A -85,B 0,C 180,E1 -5127.659,E2 -5127.659} C_VEL
LIN {X 0,Y 516.16,Z 939.786,A -85,B 0,C 180,E1 -5129.22,E2 -5129.22} C_VEL
LIN {X 0,Y 516.154,Z 940,A -85,B 0,C 180,E1 -5130,E2 -5130} C_VEL
LIN {X 0,Y 516.192,Z 939.184,A -85,B 0,C 180,E1 -5131.56,E2 -5131.56} C_VEL
LIN {X 0,Y 516.261,Z 938.197,A -85,B 0,C 180,E1 -5132.341,E2 -5132.341} C_VEL
LIN {X 0,Y 516.283,Z 936.81,A -85,B 0,C 180,E1 -5133.121,E2 -5133.121} C_VEL
LIN {X 0,Y 516.344,Z 933.895,A -85,B 0,C 180,E1 -5134.293,E2 -5134.293} C_VEL
LIN {X 0,Y 516.406,Z 929.948,A -85,B 0,C 180,E1 -5135.467,E2 -5135.467} C_VEL
LIN {X 0,Y 516.487,Z 924.033,A -85,B 0,C 180,E1 -5136.807,E2 -5136.807} C_VEL
LIN {X 0,Y 516.642,Z 917.235,A -85,B 0,C 180,E1 -5138.015,E2 -5138.015} C_VEL
LIN {X 0,Y 516.868,Z 908.991,A -85,B 0,C 180,E1 -5139.193,E2 -5139.193} C_VEL
LIN {X 0,Y 517.079,Z 900.539,A -85,B 0,C 180,E1 -5140.177,E2 -5140.177} C_VEL
LIN {X 0,Y 517.471,Z 890.092,A -85,B 0,C 180,E1 -5141.159,E2 -5141.159} C_VEL
LIN {X 0,Y 517.757,Z 878.678,A -85,B 0,C 180,E1 -5142.021,E2 -5142.021} C_VEL
LIN {X 0,Y 518.006,Z 868.404,A -85,B 0,C 180,E1 -5142.637,E2 -5142.637} C_VEL
LIN {X 0,Y 518.271,Z 856.762,A -85,B 0,C 180,E1 -5143.179,E2 -5143.179} C_VEL
LIN {X 0,Y 518.416,Z 843.685,A -85,B 0,C 180,E1 -5143.615,E2 -5143.615} C_VEL
LIN {X 0,Y 516.587,Z 832.53,A -85,B 0,C 180,E1 -5143.924,E2 -5143.924} C_VEL
LIN {X 0,Y 516.749,Z 822.435,A -85,B 0,C 180,E1 -5147.002,E2 -5147.002} C_VEL
LIN {X 0,Y 516.873,Z 814.149,A -85,B 0,C 180,E1 -5149.459,E2 -5149.459} C_VEL
LIN {X 0,Y 517.032,Z 804.043,A -85,B 0,C 180,E1 -5152.433,E2 -5152.433} C_VEL
LIN {X 0,Y 517.153,Z 794.564,A -85,B 0,C 180,E1 -5155.346,E2 -5155.346} C_VEL
LIN {X 0,Y 517.341,Z 786.169,A -85,B 0,C 180,E1 -5157.991,E2 -5157.991} C_VEL
LIN {X 0,Y 517.603,Z 776.599,A -85,B 0,C 180,E1 -5161.194,E2 -5161.194} C_VEL
LIN {X 0,Y 517.939,Z 768.625,A -85,B 0,C 180,E1 -5164.134,E2 -5164.134} C_VEL
LIN {X 0,Y 518.036,Z 763.792,A -85,B 0,C 180,E1 -5166.168,E2 -5166.168} C_VEL
LIN {X 0,Y 517.232,Z 758.924,A -85,B 0,C 180,E1 -5168.685,E2 -5168.685} C_VEL
LIN {X 0,Y 516.907,Z 757.1,A -85,B 0,C 180,E1 -5169.969,E2 -5169.969} C_VEL
LIN {X 0,Y 516.889,Z 757.102,A -85,B 0,C 180,E1 -5172.831,E2 -5172.831} C_VEL
LIN {X 0,Y 516.928,Z 757.098,A -85,B 0,C 180,E1 -5175.01,E2 -5175.01} C_VEL
LIN {X 0,Y 516.907,Z 757.098,A -85,B 0,C 180,E1 -5178.4,E2 -5178.4} C_VEL
LIN {X 0,Y 516.884,Z 757.103,A -85,B 0,C 180,E1 -5181.284,E2 -5181.284} C_VEL
LIN {X 0,Y 516.816,Z 757.11,A -85,B 0,C 180,E1 -5184.215,E2 -5184.215} C_VEL
LIN {X 0,Y 516.811,Z 757.113,A -85,B 0,C 180,E1 -5185.169,E2 -5185.169} C_VEL
LIN {X 0,Y 516.737,Z 758.78,A -85,B 0,C 180,E1 -5187.485,E2 -5187.485} C_VEL
LIN {X 0,Y 516.604,Z 761.559,A -85,B 0,C 180,E1 -5190.675,E2 -5190.675} C_VEL
LIN {X 0,Y 516.482,Z 764.488,A -85,B 0,C 180,E1 -5193.909,E2 -5193.909} C_VEL
LIN {X 0,Y 516.402,Z 767.183,A -85,B 0,C 180,E1 -5196.753,E2 -5196.753} C_VEL
LIN {X 0,Y 516.352,Z 770.212,A -85,B 0,C 180,E1 -5199.91,E2 -5199.91} C_VEL
LIN {X 0,Y 516.266,Z 772.793,A -85,B 0,C 180,E1 -5202.572,E2 -5202.572} C_VEL
LIN {X 0,Y 516.254,Z 775.421,A -85,B 0,C 180,E1 -5205.141,E2 -5205.141} C_VEL
LIN {X 0,Y 516.262,Z 776.676,A -85,B 0,C 180,E1 -5206.192,E2 -5206.192} C_VEL
LIN {X 0,Y 518.438,Z 790.097,A -85,B 0,C 180,E1 -5206.626,E2 -5206.626} C_VEL
LIN {X 0,Y 518.133,Z 802.57,A -85,B 0,C 180,E1 -5207.116,E2 -5207.116} C_VEL
LIN {X 0,Y 517.84,Z 815.304,A -85,B 0,C 180,E1 -5207.808,E2 -5207.808} C_VEL
LIN {X 0,Y 517.569,Z 827.176,A -85,B 0,C 180,E1 -5208.644,E2 -5208.644} C_VEL
LIN {X 0,Y 517.265,Z 836.174,A -85,B 0,C 180,E1 -5209.43,E2 -5209.43} C_VEL
LIN {X 0,Y 516.976,Z 845.409,A -85,B 0,C 180,E1 -5210.413,E2 -5210.413} C_VEL
LIN {X 0,Y 516.722,Z 854.373,A -85,B 0,C 180,E1 -5211.592,E2 -5211.592} C_VEL
LIN {X 0,Y 516.515,Z 861.594,A -85,B 0,C 180,E1 -5212.769,E2 -5212.769} C_VEL
LIN {X 0,Y 516.429,Z 866.468,A -85,B 0,C 180,E1 -5213.749,E2 -5213.749} C_VEL
LIN {X 0,Y 516.314,Z 871.206,A -85,B 0,C 180,E1 -5214.923,E2 -5214.923} C_VEL
LIN {X 0,Y 516.355,Z 874.836,A -85,B 0,C 180,E1 -5216.097,E2 -5216.097} C_VEL
LIN {X 0,Y 516.283,Z 876.712,A -85,B 0,C 180,E1 -5216.878,E2 -5216.878} C_VEL
LIN {X 0,Y 516.261,Z 878.131,A -85,B 0,C 180,E1 -5217.659,E2 -5217.659} C_VEL
LIN {X 0,Y 516.161,Z 879.758,A -85,B 0,C 180,E1 -5219.219,E2 -5219.219} C_VEL
LIN {X 0,Y 516.154,Z 879.997,A -85,B 0,C 180,E1 -5219.999,E2 -5219.999} C_VEL
LIN {X 0,Y 516.16,Z 879.813,A -85,B 0,C 180,E1 -5220.779,E2 -5220.779} C_VEL
LIN {X 0,Y 516.261,Z 878.26,A -85,B 0,C 180,E1 -5222.34,E2 -5222.34} C_VEL
LIN {X 0,Y 516.283,Z 876.898,A -85,B 0,C 180,E1 -5223.121,E2 -5223.121} C_VEL
LIN {X 0,Y 516.344,Z 874.019,A -85,B 0,C 180,E1 -5224.292,E2 -5224.292} C_VEL
LIN {X 0,Y 516.4,Z 870.116,A -85,B 0,C 180,E1 -5225.466,E2 -5225.466} C_VEL
LIN {X 0,Y 516.476,Z 864.328,A -85,B 0,C 180,E1 -5226.795,E2 -5226.795} C_VEL
LIN {X 0,Y 516.64,Z 857.522,A -85,B 0,C 180,E1 -5228.014,E2 -5228.014} C_VEL
LIN {X 0,Y 516.865,Z 849.338,A -85,B 0,C 180,E1 -5229.193,E2 -5229.193} C_VEL
LIN {X 0,Y 517.071,Z 840.965,A -85,B 0,C 180,E1 -5230.176,E2 -5230.176} C_VEL
LIN {X 0,Y 517.434,Z 830.636,A -85,B 0,C 180,E1 -5231.159,E2 -5231.159} C_VEL
LIN {X 0,Y 517.697,Z 819.439,A -85,B 0,C 180,E1 -5232.015,E2 -5232.015} C_VEL
LIN {X 0,Y 518.003,Z 807.402,A -85,B 0,C 180,E1 -5232.736,E2 -5232.736} C_VEL
LIN {X 0,Y 518.311,Z 795.371,A -85,B 0,C 180,E1 -5233.276,E2 -5233.276} C_VEL
LIN {X 0,Y 518.202,Z 787.951,A -85,B 0,C 180,E1 -5233.541,E2 -5233.541} C_VEL
LIN {X 0,Y 516.246,Z 776.665,A -85,B 0,C 180,E1 -5233.907,E2 -5233.907} C_VEL
LIN {X 0,Y 516.261,Z 772.528,A -85,B 0,C 180,E1 -5237.426,E2 -5237.426} C_VEL
LIN {X 0,Y 516.297,Z 768.963,A -85,B 0,C 180,E1 -5240.726,E2 -5240.726} C_VEL
LIN {X 0,Y 516.353,Z 766.362,A -85,B 0,C 180,E1 -5243.247,E2 -5243.247} C_VEL
LIN {X 0,Y 516.383,Z 763.411,A -85,B 0,C 180,E1 -5246.069,E2 -5246.069} C_VEL
LIN {X 0,Y 516.388,Z 760.828,A -85,B 0,C 180,E1 -5248.446,E2 -5248.446} C_VEL
LIN {X 0,Y 516.456,Z 757.982,A -85,B 0,C 180,E1 -5251.137,E2 -5251.137} C_VEL
LIN {X 0,Y 516.471,Z 757.156,A -85,B 0,C 180,E1 -5252.052,E2 -5252.052} C_VEL
LIN {X 0,Y 516.805,Z 757.113,A -85,B 0,C 180,E1 -5254.83,E2 -5254.83} C_VEL
LIN {X 0,Y 516.875,Z 757.098,A -85,B 0,C 180,E1 -5257.942,E2 -5257.942} C_VEL
LIN {X 0,Y 516.879,Z 757.098,A -85,B 0,C 180,E1 -5260.741,E2 -5260.741} C_VEL
LIN {X 0,Y 516.872,Z 757.099,A -85,B 0,C 180,E1 -5262.906,E2 -5262.906} C_VEL
LIN {X 0,Y 516.918,Z 757.096,A -85,B 0,C 180,E1 -5265.009,E2 -5265.009} C_VEL
LIN {X 0,Y 516.864,Z 757.098,A -85,B 0,C 180,E1 -5266.304,E2 -5266.304} C_VEL
LIN {X 0,Y 516.187,Z 757.187,A -85,B 0,C 180,E1 -5266.955,E2 -5266.955} C_VEL
LIN {X 0,Y 513.352,Z 757.543,A -85,B 0,C 180,E1 -5268.012,E2 -5268.012} C_VEL
LIN {X 0,Y 510.955,Z 757.843,A -85,B 0,C 180,E1 -5268.864,E2 -5268.864} C_VEL
LIN {X 0,Y 509.915,Z 757.97,A -85,B 0,C 180,E1 -5269.521,E2 -5269.521} C_VEL
LIN {X 0,Y 509.823,Z 757.979,A -85,B 0,C 180,E1 -5269.743,E2 -5269.743} C_VEL
LIN {X 0,Y 509.809,Z 757.977,A -85,B 0,C 180,E1 -5272.658,E2 -5272.658} C_VEL
LIN {X 0,Y 509.835,Z 757.978,A -85,B 0,C 180,E1 -5275.799,E2 -5275.799} C_VEL
LIN {X 0,Y 509.837,Z 757.974,A -85,B 0,C 180,E1 -5278.72,E2 -5278.72} C_VEL
LIN {X 0,Y 509.845,Z 757.975,A -85,B 0,C 180,E1 -5281.154,E2 -5281.154} C_VEL
LIN {X 0,Y 509.86,Z 757.975,A -85,B 0,C 180,E1 -5283.826,E2 -5283.826} C_VEL
LIN {X 0,Y 509.81,Z 757.977,A -85,B 0,C 180,E1 -5286.435,E2 -5286.435} C_VEL
LIN {X 0,Y 509.907,Z 757.97,A -85,B 0,C 180,E1 -5289.844,E2 -5289.844} C_VEL
LIN {X 0,Y 509.857,Z 757.972,A -85,B 0,C 180,E1 -5293.174,E2 -5293.174} C_VEL
LIN {X 0,Y 509.85,Z 757.978,A -85,B 0,C 180,E1 -5295.634,E2 -5295.634} C_VEL
LIN {X 0,Y 509.9,Z 757.965,A -85,B 0,C 180,E1 -5298.874,E2 -5298.874} C_VEL
LIN {X 0,Y 509.866,Z 757.975,A -85,B 0,C 180,E1 -5302.077,E2 -5302.077} C_VEL
LIN {X 0,Y 509.926,Z 757.963,A -85,B 0,C 180,E1 -5304.464,E2 -5304.464} C_VEL
LIN {X 0,Y 510.03,Z 757.952,A -85,B 0,C 180,E1 -5307.631,E2 -5307.631} C_VEL
LIN {X 0,Y 510.023,Z 757.958,A -85,B 0,C 180,E1 -5310,E2 -5310} C_VEL
LIN {X 0,Y 510.028,Z 757.953,A -85,B 0,C 180,E1 -5312.369,E2 -5312.369} C_VEL
LIN {X 0,Y 509.923,Z 757.963,A -85,B 0,C 180,E1 -5315.536,E2 -5315.536} C_VEL
LIN {X 0,Y 509.863,Z 757.974,A -85,B 0,C 180,E1 -5317.923,E2 -5317.923} C_VEL
LIN {X 0,Y 509.849,Z 757.971,A -85,B 0,C 180,E1 -5321.127,E2 -5321.127} C_VEL
LIN {X 0,Y 509.841,Z 757.973,A -85,B 0,C 180,E1 -5323.553,E2 -5323.553} C_VEL
LIN {X 0,Y 509.827,Z 757.978,A -85,B 0,C 180,E1 -5326.004,E2 -5326.004} C_VEL
LIN {X 0,Y 509.828,Z 757.981,A -85,B 0,C 180,E1 -5328.485,E2 -5328.485} C_VEL
LIN {X 0,Y 509.841,Z 757.973,A -85,B 0,C 180,E1 -5331.002,E2 -5331.002} C_VEL
LIN {X 0,Y 509.809,Z 757.976,A -85,B 0,C 180,E1 -5333.565,E2 -5333.565} C_VEL
LIN {X 0,Y 509.828,Z 757.981,A -85,B 0,C 180,E1 -5336.362,E2 -5336.362} C_VEL
LIN {X 0,Y 509.841,Z 757.976,A -85,B 0,C 180,E1 -5338.847,E2 -5338.847} C_VEL
LIN {X 0,Y 509.81,Z 757.976,A -85,B 0,C 180,E1 -5341.591,E2 -5341.591} C_VEL
LIN {X 0,Y 509.83,Z 757.979,A -85,B 0,C 180,E1 -5344.415,E2 -5344.415} C_VEL
LIN {X 0,Y 509.809,Z 757.977,A -85,B 0,C 180,E1 -5347.342,E2 -5347.342} C_VEL
LIN {X 0,Y 509.831,Z 757.978,A -85,B 0,C 180,E1 -5350.383,E2 -5350.383} C_VEL
LIN {X 0,Y 509.816,Z 757.98,A -85,B 0,C 180,E1 -5353.063,E2 -5353.063} C_VEL
LIN {X 0,Y 509.817,Z 757.976,A -85,B 0,C 180,E1 -5355.794,E2 -5355.794} C_VEL
LIN {X 0,Y 509.85,Z 757.977,A -85,B 0,C 180,E1 -5358.575,E2 -5358.575} C_VEL
LIN {X 0,Y 509.846,Z 757.972,A -85,B 0,C 180,E1 -5361.788,E2 -5361.788} C_VEL
LIN {X 0,Y 509.782,Z 757.985,A -85,B 0,C 180,E1 -5364.619,E2 -5364.619} C_VEL
LIN {X 0,Y 509.545,Z 758.017,A -85,B 0,C 180,E1 -5367.459,E2 -5367.459} C_VEL
LIN {X 0,Y 509.374,Z 758.038,A -85,B 0,C 180,E1 -5368.808,E2 -5368.808} C_VEL
LIN {X 0,Y 509.277,Z 759.547,A -85,B 0,C 180,E1 -5370.389,E2 -5370.389} C_VEL
LIN {X 0,Y 509.301,Z 762.44,A -85,B 0,C 180,E1 -5372.912,E2 -5372.912} C_VEL
LIN {X 0,Y 509.269,Z 765.422,A -85,B 0,C 180,E1 -5375.618,E2 -5375.618} C_VEL
LIN {X 0,Y 509.241,Z 768.21,A -85,B 0,C 180,E1 -5378.123,E2 -5378.123} C_VEL
LIN {X 0,Y 509.172,Z 771.057,A -85,B 0,C 180,E1 -5380.655,E2 -5380.655} C_VEL
LIN {X 0,Y 509.168,Z 773.707,A -85,B 0,C 180,E1 -5383.151,E2 -5383.151} C_VEL
LIN {X 0,Y 509.181,Z 776.813,A -85,B 0,C 180,E1 -5385.998,E2 -5385.998} C_VEL
LIN {X 0,Y 511.459,Z 790.198,A -85,B 0,C 180,E1 -5386.441,E2 -5386.441} C_VEL
LIN {X 0,Y 511.171,Z 802.426,A -85,B 0,C 180,E1 -5386.939,E2 -5386.939} C_VEL
LIN {X 0,Y 510.911,Z 812.034,A -85,B 0,C 180,E1 -5387.445,E2 -5387.445} C_VEL
LIN {X 0,Y 510.72,Z 821.846,A -85,B 0,C 180,E1 -5388.089,E2 -5388.089} C_VEL
LIN {X 0,Y 510.449,Z 830.652,A -85,B 0,C 180,E1 -5388.787,E2 -5388.787} C_VEL
LIN {X 0,Y 510.185,Z 838.117,A -85,B 0,C 180,E1 -5389.484,E2 -5389.484} C_VEL
LIN {X 0,Y 509.971,Z 845.39,A -85,B 0,C 180,E1 -5390.282,E2 -5390.282} C_VEL
LIN {X 0,Y 509.742,Z 852.979,A -85,B 0,C 180,E1 -5391.278,E2 -5391.278} C_VEL
LIN {X 0,Y 509.523,Z 859.313,A -85,B 0,C 180,E1 -5392.272,E2 -5392.272} C_VEL
LIN {X 0,Y 509.367,Z 865.33,A -85,B 0,C 180,E1 -5393.426,E2 -5393.426} C_VEL
LIN {X 0,Y 509.345,Z 869.714,A -85,B 0,C 180,E1 -5394.458,E2 -5394.458} C_VEL
LIN {X 0,Y 509.233,Z 873.693,A -85,B 0,C 180,E1 -5395.648,E2 -5395.648} C_VEL
LIN {X 0,Y 509.2,Z 876.642,A -85,B 0,C 180,E1 -5396.836,E2 -5396.836} C_VEL
LIN {X 0,Y 509.161,Z 878.146,A -85,B 0,C 180,E1 -5397.628,E2 -5397.628} C_VEL
LIN {X 0,Y 509.074,Z 879.708,A -85,B 0,C 180,E1 -5399.21,E2 -5399.21} C_VEL
LIN {X 0,Y 509.065,Z 879.999,A -85,B 0,C 180,E1 -5400.001,E2 -5400.001} C_VEL
LIN {X 0,Y 509.112,Z 879.187,A -85,B 0,C 180,E1 -5401.583,E2 -5401.583} C_VEL
LIN {X 0,Y 509.161,Z 878.279,A -85,B 0,C 180,E1 -5402.374,E2 -5402.374} C_VEL
LIN {X 0,Y 509.254,Z 875.023,A -85,B 0,C 180,E1 -5403.957,E2 -5403.957} C_VEL
LIN {X 0,Y 509.247,Z 871.463,A -85,B 0,C 180,E1 -5405.147,E2 -5405.147} C_VEL
LIN {X 0,Y 509.36,Z 868.571,A -85,B 0,C 180,E1 -5405.941,E2 -5405.941} C_VEL
LIN {X 0,Y 509.424,Z 863.088,A -85,B 0,C 180,E1 -5407.133,E2 -5407.133} C_VEL
LIN {X 0,Y 509.621,Z 856.206,A -85,B 0,C 180,E1 -5408.327,E2 -5408.327} C_VEL
LIN {X 0,Y 509.806,Z 849.238,A -85,B 0,C 180,E1 -5409.323,E2 -5409.323} C_VEL
LIN {X 0,Y 510.015,Z 842.677,A -85,B 0,C 180,E1 -5410.12,E2 -5410.12} C_VEL
LIN {X 0,Y 510.34,Z 833.852,A -85,B 0,C 180,E1 -5411.016,E2 -5411.016} C_VEL
LIN {X 0,Y 510.607,Z 825.677,A -85,B 0,C 180,E1 -5411.714,E2 -5411.714} C_VEL
LIN {X 0,Y 510.813,Z 816.788,A -85,B 0,C 180,E1 -5412.351,E2 -5412.351} C_VEL
LIN {X 0,Y 511.087,Z 807.206,A -85,B 0,C 180,E1 -5412.913,E2 -5412.913} C_VEL
LIN {X 0,Y 511.332,Z 797.684,A -85,B 0,C 180,E1 -5413.361,E2 -5413.361} C_VEL
LIN {X 0,Y 511.284,Z 789.096,A -85,B 0,C 180,E1 -5413.692,E2 -5413.692} C_VEL
LIN {X 0,Y 509.17,Z 776.944,A -85,B 0,C 180,E1 -5414.081,E2 -5414.081} C_VEL
LIN {X 0,Y 509.171,Z 774.083,A -85,B 0,C 180,E1 -5416.85,E2 -5416.85} C_VEL
LIN {X 0,Y 509.185,Z 771.426,A -85,B 0,C 180,E1 -5419.346,E2 -5419.346} C_VEL
LIN {X 0,Y 509.287,Z 768.06,A -85,B 0,C 180,E1 -5422.395,E2 -5422.395} C_VEL
LIN {X 0,Y 509.293,Z 764.732,A -85,B 0,C 180,E1 -5425.328,E2 -5425.328} C_VEL
LIN {X 0,Y 509.288,Z 761.396,A -85,B 0,C 180,E1 -5427.982,E2 -5427.982} C_VEL
LIN {X 0,Y 509.257,Z 759.012,A -85,B 0,C 180,E1 -5429.79,E2 -5429.79} C_VEL
LIN {X 0,Y 509.26,Z 758.054,A -85,B 0,C 180,E1 -5430.705,E2 -5430.705} C_VEL
LIN {X 0,Y 509.602,Z 758.011,A -85,B 0,C 180,E1 -5433.481,E2 -5433.481} C_VEL
LIN {X 0,Y 509.777,Z 757.986,A -85,B 0,C 180,E1 -5435.57,E2 -5435.57} C_VEL
LIN {X 0,Y 509.854,Z 757.972,A -85,B 0,C 180,E1 -5438.338,E2 -5438.338} C_VEL
LIN {X 0,Y 509.855,Z 757.976,A -85,B 0,C 180,E1 -5441.426,E2 -5441.426} C_VEL
LIN {X 0,Y 509.862,Z 757.975,A -85,B 0,C 180,E1 -5444.668,E2 -5444.668} C_VEL
LIN {X 0,Y 509.86,Z 757.972,A -85,B 0,C 180,E1 -5448.104,E2 -5448.104} C_VEL
LIN {X 0,Y 509.881,Z 758.127,A -85,B 0,C 180,E1 -5450.969,E2 -5450.969} C_VEL
LIN {X 0,Y 511.077,Z 765.055,A -85,B 0,C 180,E1 -5453.75,E2 -5453.75} C_VEL
LIN {X 0,Y 511.132,Z 770.25,A -85,B 0,C 180,E1 -5455.685,E2 -5455.685} C_VEL
LIN {X 0,Y 510.824,Z 778.23,A -85,B 0,C 180,E1 -5458.541,E2 -5458.541} C_VEL
LIN {X 0,Y 510.546,Z 785.974,A -85,B 0,C 180,E1 -5461.197,E2 -5461.197} C_VEL
LIN {X 0,Y 510.309,Z 793.916,A -85,B 0,C 180,E1 -5463.851,E2 -5463.851} C_VEL
LIN {X 0,Y 510.089,Z 803.285,A -85,B 0,C 180,E1 -5466.879,E2 -5466.879} C_VEL
LIN {X 0,Y 509.848,Z 814.069,A -85,B 0,C 180,E1 -5470.262,E2 -5470.262} C_VEL
LIN {X 0,Y 509.653,Z 823.596,A -85,B 0,C 180,E1 -5473.167,E2 -5473.167} C_VEL
LIN {X 0,Y 509.554,Z 832.725,A -85,B 0,C 180,E1 -5475.899,E2 -5475.899} C_VEL
LIN {X 0,Y 511.591,Z 845.179,A -85,B 0,C 180,E1 -5476.241,E2 -5476.241} C_VEL
LIN {X 0,Y 511.353,Z 857.979,A -85,B 0,C 180,E1 -5476.69,E2 -5476.69} C_VEL
LIN {X 0,Y 511.012,Z 870.17,A -85,B 0,C 180,E1 -5477.288,E2 -5477.288} C_VEL
LIN {X 0,Y 510.711,Z 880.935,A -85,B 0,C 180,E1 -5477.97,E2 -5477.97} C_VEL
LIN {X 0,Y 510.41,Z 892.397,A -85,B 0,C 180,E1 -5478.885,E2 -5478.885} C_VEL
LIN {X 0,Y 510.035,Z 902.332,A -85,B 0,C 180,E1 -5479.881,E2 -5479.881} C_VEL
LIN {X 0,Y 509.761,Z 911.96,A -85,B 0,C 180,E1 -5481.077,E2 -5481.077} C_VEL
LIN {X 0,Y 509.523,Z 919.621,A -85,B 0,C 180,E1 -5482.271,E2 -5482.271} C_VEL
LIN {X 0,Y 509.337,Z 926.679,A -85,B 0,C 180,E1 -5483.662,E2 -5483.662} C_VEL
LIN {X 0,Y 509.248,Z 931.373,A -85,B 0,C 180,E1 -5484.853,E2 -5484.853} C_VEL
LIN {X 0,Y 509.254,Z 934.958,A -85,B 0,C 180,E1 -5486.043,E2 -5486.043} C_VEL
LIN {X 0,Y 509.201,Z 936.807,A -85,B 0,C 180,E1 -5486.835,E2 -5486.835} C_VEL
LIN {X 0,Y 509.161,Z 938.194,A -85,B 0,C 180,E1 -5487.627,E2 -5487.627} C_VEL
LIN {X 0,Y 509.074,Z 939.786,A -85,B 0,C 180,E1 -5489.209,E2 -5489.209} C_VEL
LIN {X 0,Y 509.065,Z 940,A -85,B 0,C 180,E1 -5490,E2 -5490} C_VEL
LIN {X 0,Y 509.113,Z 939.184,A -85,B 0,C 180,E1 -5491.582,E2 -5491.582} C_VEL
LIN {X 0,Y 509.161,Z 938.196,A -85,B 0,C 180,E1 -5492.373,E2 -5492.373} C_VEL
LIN {X 0,Y 509.201,Z 936.81,A -85,B 0,C 180,E1 -5493.165,E2 -5493.165} C_VEL
LIN {X 0,Y 509.234,Z 933.895,A -85,B 0,C 180,E1 -5494.353,E2 -5494.353} C_VEL
LIN {X 0,Y 509.345,Z 929.948,A -85,B 0,C 180,E1 -5495.543,E2 -5495.543} C_VEL
LIN {X 0,Y 509.411,Z 924.281,A -85,B 0,C 180,E1 -5496.853,E2 -5496.853} C_VEL
LIN {X 0,Y 509.586,Z 917.235,A -85,B 0,C 180,E1 -5498.127,E2 -5498.127} C_VEL
LIN {X 0,Y 509.847,Z 908.992,A -85,B 0,C 180,E1 -5499.321,E2 -5499.321} C_VEL
LIN {X 0,Y 510.067,Z 900.539,A -85,B 0,C 180,E1 -5500.319,E2 -5500.319} C_VEL
LIN {X 0,Y 510.503,Z 890.091,A -85,B 0,C 180,E1 -5501.314,E2 -5501.314} C_VEL
LIN {X 0,Y 510.789,Z 879.419,A -85,B 0,C 180,E1 -5502.135,E2 -5502.135} C_VEL
LIN {X 0,Y 511.068,Z 868.403,A -85,B 0,C 180,E1 -5502.812,E2 -5502.812} C_VEL
LIN {X 0,Y 511.378,Z 856.762,A -85,B 0,C 180,E1 -5503.359,E2 -5503.359} C_VEL
LIN {X 0,Y 511.467,Z 844.256,A -85,B 0,C 180,E1 -5503.787,E2 -5503.787} C_VEL
LIN {X 0,Y 509.543,Z 832.53,A -85,B 0,C 180,E1 -5504.12,E2 -5504.12} C_VEL
LIN {X 0,Y 509.644,Z 823.448,A -85,B 0,C 180,E1 -5506.834,E2 -5506.834} C_VEL
LIN {X 0,Y 509.778,Z 815.044,A -85,B 0,C 180,E1 -5509.322,E2 -5509.322} C_VEL
LIN {X 0,Y 509.952,Z 805.37,A -85,B 0,C 180,E1 -5512.215,E2 -5512.215} C_VEL
LIN {X 0,Y 510.113,Z 795.536,A -85,B 0,C 180,E1 -5515.284,E2 -5515.284} C_VEL
LIN {X 0,Y 510.314,Z 786.496,A -85,B 0,C 180,E1 -5518.187,E2 -5518.187} C_VEL
LIN {X 0,Y 510.637,Z 777.114,A -85,B 0,C 180,E1 -5521.425,E2 -5521.425} C_VEL
LIN {X 0,Y 510.9,Z 770.665,A -85,B 0,C 180,E1 -5523.857,E2 -5523.857} C_VEL
LIN {X 0,Y 511.104,Z 766.091,A -85,B 0,C 180,E1 -5525.777,E2 -5525.777} C_VEL
LIN {X 0,Y 510.758,Z 763.037,A -85,B 0,C 180,E1 -5527.261,E2 -5527.261} C_VEL
LIN {X 0,Y 509.924,Z 758.291,A -85,B 0,C 180,E1 -5530.136,E2 -5530.136} C_VEL
LIN {X 0,Y 509.843,Z 757.98,A -85,B 0,C 180,E1 -5530.698,E2 -5530.698} C_VEL
LIN {X 0,Y 509.825,Z 757.982,A -85,B 0,C 180,E1 -5533.572,E2 -5533.572} C_VEL
LIN {X 0,Y 509.816,Z 757.982,A -85,B 0,C 180,E1 -5536.427,E2 -5536.427} C_VEL
LIN {X 0,Y 509.834,Z 757.981,A -85,B 0,C 180,E1 -5539.303,E2 -5539.303} C_VEL
LIN {X 0,Y 509.854,Z 757.976,A -85,B 0,C 180,E1 -5541.786,E2 -5541.786} C_VEL
LIN {X 0,Y 509.784,Z 757.988,A -85,B 0,C 180,E1 -5544.618,E2 -5544.618} C_VEL
LIN {X 0,Y 509.778,Z 758.429,A -85,B 0,C 180,E1 -5545.811,E2 -5545.811} C_VEL
LIN {X 0,Y 509.617,Z 760.816,A -85,B 0,C 180,E1 -5548.763,E2 -5548.763} C_VEL
LIN {X 0,Y 509.512,Z 762.846,A -85,B 0,C 180,E1 -5551.132,E2 -5551.132} C_VEL
LIN {X 0,Y 509.457,Z 765.224,A -85,B 0,C 180,E1 -5553.803,E2 -5553.803} C_VEL
LIN {X 0,Y 509.342,Z 767.639,A -85,B 0,C 180,E1 -5556.412,E2 -5556.412} C_VEL
LIN {X 0,Y 509.31,Z 770.131,A -85,B 0,C 180,E1 -5558.974,E2 -5558.974} C_VEL
LIN {X 0,Y 509.233,Z 773.304,A -85,B 0,C 180,E1 -5562.324,E2 -5562.324} C_VEL
LIN {X 0,Y 509.162,Z 776.801,A -85,B 0,C 180,E1 -5565.817,E2 -5565.817} C_VEL
LIN {X 0,Y 509.182,Z 776.983,A -85,B 0,C 180,E1 -5565.996,E2 -5565.996} C_VEL
LIN {X 0,Y 511.507,Z 790.887,A -85,B 0,C 180,E1 -5566.466,E2 -5566.466} C_VEL
LIN {X 0,Y 511.182,Z 803.597,A -85,B 0,C 180,E1 -5566.989,E2 -5566.989} C_VEL
LIN {X 0,Y 510.879,Z 815.744,A -85,B 0,C 180,E1 -5567.667,E2 -5567.667} C_VEL
LIN {X 0,Y 510.603,Z 827.185,A -85,B 0,C 180,E1 -5568.487,E2 -5568.487} C_VEL
LIN {X 0,Y 510.264,Z 836.181,A -85,B 0,C 180,E1 -5569.283,E2 -5569.283} C_VEL
LIN {X 0,Y 509.973,Z 845.414,A -85,B 0,C 180,E1 -5570.28,E2 -5570.28} C_VEL
LIN {X 0,Y 509.677,Z 854.377,A -85,B 0,C 180,E1 -5571.475,E2 -5571.475} C_VEL
LIN {X 0,Y 509.442,Z 861.597,A -85,B 0,C 180,E1 -5572.668,E2 -5572.668} C_VEL
LIN {X 0,Y 509.369,Z 868.179,A -85,B 0,C 180,E1 -5574.06,E2 -5574.06} C_VEL
LIN {X 0,Y 509.189,Z 872.533,A -85,B 0,C 180,E1 -5575.249,E2 -5575.249} C_VEL
LIN {X 0,Y 509.254,Z 874.837,A -85,B 0,C 180,E1 -5576.043,E2 -5576.043} C_VEL
LIN {X 0,Y 509.201,Z 876.713,A -85,B 0,C 180,E1 -5576.834,E2 -5576.834} C_VEL
LIN {X 0,Y 509.161,Z 878.131,A -85,B 0,C 180,E1 -5577.626,E2 -5577.626} C_VEL
LIN {X 0,Y 509.074,Z 879.758,A -85,B 0,C 180,E1 -5579.208,E2 -5579.208} C_VEL
LIN {X 0,Y 509.065,Z 879.997,A -85,B 0,C 180,E1 -5579.999,E2 -5579.999} C_VEL
LIN {X 0,Y 509.074,Z 879.813,A -85,B 0,C 180,E1 -5580.79,E2 -5580.79} C_VEL
LIN {X 0,Y 509.161,Z 878.258,A -85,B 0,C 180,E1 -5582.372,E2 -5582.372} C_VEL
LIN {X 0,Y 509.201,Z 876.896,A -85,B 0,C 180,E1 -5583.164,E2 -5583.164} C_VEL
LIN {X 0,Y 509.233,Z 874.017,A -85,B 0,C 180,E1 -5584.352,E2 -5584.352} C_VEL
LIN {X 0,Y 509.337,Z 870.114,A -85,B 0,C 180,E1 -5585.542,E2 -5585.542} C_VEL
LIN {X 0,Y 509.383,Z 865.08,A -85,B 0,C 180,E1 -5586.734,E2 -5586.734} C_VEL
LIN {X 0,Y 509.565,Z 858.746,A -85,B 0,C 180,E1 -5587.927,E2 -5587.927} C_VEL
LIN {X 0,Y 509.78,Z 850.818,A -85,B 0,C 180,E1 -5589.121,E2 -5589.121} C_VEL
LIN {X 0,Y 510.017,Z 842.74,A -85,B 0,C 180,E1 -5590.118,E2 -5590.118} C_VEL
LIN {X 0,Y 510.396,Z 832.886,A -85,B 0,C 180,E1 -5591.114,E2 -5591.114} C_VEL
LIN {X 0,Y 510.709,Z 823.198,A -85,B 0,C 180,E1 -5591.912,E2 -5591.912} C_VEL
LIN {X 0,Y 510.955,Z 812.263,A -85,B 0,C 180,E1 -5592.639,E2 -5592.639} C_VEL
LIN {X 0,Y 511.263,Z 800.135,A -85,B 0,C 180,E1 -5593.26,E2 -5593.26} C_VEL
LIN {X 0,Y 511.264,Z 788.704,A -85,B 0,C 180,E1 -5593.703,E2 -5593.703} C_VEL
LIN {X 0,Y 509.144,Z 776.766,A -85,B 0,C 180,E1 -5594.105,E2 -5594.105} C_VEL
LIN {X 0,Y 509.166,Z 773.734,A -85,B 0,C 180,E1 -5596.849,E2 -5596.849} C_VEL
LIN {X 0,Y 509.239,Z 770.156,A -85,B 0,C 180,E1 -5600.204,E2 -5600.204} C_VEL
LIN {X 0,Y 509.264,Z 767.568,A -85,B 0,C 180,E1 -5602.73,E2 -5602.73} C_VEL
LIN {X 0,Y 509.288,Z 764.757,A -85,B 0,C 180,E1 -5605.326,E2 -5605.326} C_VEL
LIN {X 0,Y 509.321,Z 761.952,A -85,B 0,C 180,E1 -5607.978,E2 -5607.978} C_VEL
LIN {X 0,Y 509.37,Z 759.074,A -85,B 0,C 180,E1 -5610.696,E2 -5610.696} C_VEL
LIN {X 0,Y 509.39,Z 758.125,A -85,B 0,C 180,E1 -5611.619,E2 -5611.619} C_VEL
LIN {X 0,Y 509.716,Z 757.996,A -85,B 0,C 180,E1 -5614.423,E2 -5614.423} C_VEL
LIN {X 0,Y 509.804,Z 757.983,A -85,B 0,C 180,E1 -5617.341,E2 -5617.341} C_VEL
LIN {X 0,Y 509.834,Z 757.974,A -85,B 0,C 180,E1 -5620.381,E2 -5620.381} C_VEL
LIN {X 0,Y 509.818,Z 757.981,A -85,B 0,C 180,E1 -5623.061,E2 -5623.061} C_VEL
LIN {X 0,Y 509.826,Z 757.978,A -85,B 0,C 180,E1 -5625.791,E2 -5625.791} C_VEL
LIN {X 0,Y 509.849,Z 757.972,A -85,B 0,C 180,E1 -5628.574,E2 -5628.574} C_VEL
LIN {X 0,Y 509.823,Z 757.979,A -85,B 0,C 180,E1 -5629.743,E2 -5629.743} C_VEL
LIN {X 0,Y 509.141,Z 758.061,A -85,B 0,C 180,E1 -5630.403,E2 -5630.403} C_VEL
LIN {X 0,Y 506.292,Z 758.421,A -85,B 0,C 180,E1 -5631.474,E2 -5631.474} C_VEL
LIN {X 0,Y 503.887,Z 758.721,A -85,B 0,C 180,E1 -5632.338,E2 -5632.338} C_VEL
LIN {X 0,Y 502.845,Z 758.848,A -85,B 0,C 180,E1 -5633.004,E2 -5633.004} C_VEL
LIN {X 0,Y 502.755,Z 758.857,A -85,B 0,C 180,E1 -5633.23,E2 -5633.23} C_VEL
LIN {X 0,Y 502.781,Z 758.855,A -85,B 0,C 180,E1 -5636.004,E2 -5636.004} C_VEL
LIN {X 0,Y 502.786,Z 758.852,A -85,B 0,C 180,E1 -5638.856,E2 -5638.856} C_VEL
LIN {X 0,Y 502.79,Z 758.857,A -85,B 0,C 180,E1 -5641.714,E2 -5641.714} C_VEL
LIN {X 0,Y 502.782,Z 758.853,A -85,B 0,C 180,E1 -5644.321,E2 -5644.321} C_VEL
LIN {X 0,Y 502.794,Z 758.854,A -85,B 0,C 180,E1 -5647.297,E2 -5647.297} C_VEL
LIN {X 0,Y 502.81,Z 758.849,A -85,B 0,C 180,E1 -5650.399,E2 -5650.399} C_VEL
LIN {X 0,Y 502.802,Z 758.849,A -85,B 0,C 180,E1 -5652.93,E2 -5652.93} C_VEL
LIN {X 0,Y 502.832,Z 758.849,A -85,B 0,C 180,E1 -5655.429,E2 -5655.429} C_VEL
LIN {X 0,Y 502.865,Z 758.841,A -85,B 0,C 180,E1 -5658.716,E2 -5658.716} C_VEL
LIN {X 0,Y 502.838,Z 758.852,A -85,B 0,C 180,E1 -5661.966,E2 -5661.966} C_VEL
LIN {X 0,Y 502.883,Z 758.842,A -85,B 0,C 180,E1 -5664.386,E2 -5664.386} C_VEL
LIN {X 0,Y 502.998,Z 758.828,A -85,B 0,C 180,E1 -5667.598,E2 -5667.598} C_VEL
LIN {X 0,Y 502.992,Z 758.834,A -85,B 0,C 180,E1 -5670,E2 -5670} C_VEL
LIN {X 0,Y 502.995,Z 758.828,A -85,B 0,C 180,E1 -5672.402,E2 -5672.402} C_VEL
LIN {X 0,Y 502.88,Z 758.841,A -85,B 0,C 180,E1 -5675.614,E2 -5675.614} C_VEL
LIN {X 0,Y 502.835,Z 758.851,A -85,B 0,C 180,E1 -5678.034,E2 -5678.034} C_VEL
LIN {X 0,Y 502.825,Z 758.846,A -85,B 0,C 180,E1 -5681.284,E2 -5681.284} C_VEL
LIN {X 0,Y 502.831,Z 758.85,A -85,B 0,C 180,E1 -5684.571,E2 -5684.571} C_VEL
LIN {X 0,Y 502.791,Z 758.853,A -85,B 0,C 180,E1 -5687.91,E2 -5687.91} C_VEL
LIN {X 0,Y 502.82,Z 758.853,A -85,B 0,C 180,E1 -5690.537,E2 -5690.537} C_VEL
LIN {X 0,Y 502.777,Z 758.853,A -85,B 0,C 180,E1 -5693.041,E2 -5693.041} C_VEL
LIN {X 0,Y 502.77,Z 758.854,A -85,B 0,C 180,E1 -5695.68,E2 -5695.68} C_VEL
LIN {X 0,Y 502.787,Z 758.857,A -85,B 0,C 180,E1 -5698.376,E2 -5698.376} C_VEL
LIN {X 0,Y 502.786,Z 758.853,A -85,B 0,C 180,E1 -5701.144,E2 -5701.144} C_VEL
LIN {X 0,Y 502.781,Z 758.854,A -85,B 0,C 180,E1 -5703.996,E2 -5703.996} C_VEL
LIN {X 0,Y 502.77,Z 758.856,A -85,B 0,C 180,E1 -5707.178,E2 -5707.178} C_VEL
LIN {X 0,Y 502.781,Z 758.854,A -85,B 0,C 180,E1 -5710.016,E2 -5710.016} C_VEL
LIN {X 0,Y 502.797,Z 758.853,A -85,B 0,C 180,E1 -5712.2,E2 -5712.2} C_VEL
LIN {X 0,Y 502.78,Z 758.853,A -85,B 0,C 180,E1 -5715.471,E2 -5715.471} C_VEL
LIN {X 0,Y 502.815,Z 758.856,A -85,B 0,C 180,E1 -5718.935,E2 -5718.935} C_VEL
LIN {X 0,Y 502.788,Z 758.852,A -85,B 0,C 180,E1 -5722.047,E2 -5722.047} C_VEL
LIN {X 0,Y 502.693,Z 758.871,A -85,B 0,C 180,E1 -5725.027,E2 -5725.027} C_VEL
LIN {X 0,Y 502.43,Z 758.904,A -85,B 0,C 180,E1 -5727.891,E2 -5727.891} C_VEL
LIN {X 0,Y 502.349,Z 758.913,A -85,B 0,C 180,E1 -5728.827,E2 -5728.827} C_VEL
LIN {X 0,Y 502.201,Z 759.913,A -85,B 0,C 180,E1 -5730.187,E2 -5730.187} C_VEL
LIN {X 0,Y 502.267,Z 763.765,A -85,B 0,C 180,E1 -5733.576,E2 -5733.576} C_VEL
LIN {X 0,Y 502.182,Z 766.469,A -85,B 0,C 180,E1 -5736.057,E2 -5736.057} C_VEL
LIN {X 0,Y 502.153,Z 769.338,A -85,B 0,C 180,E1 -5738.662,E2 -5738.662} C_VEL
LIN {X 0,Y 502.08,Z 772.189,A -85,B 0,C 180,E1 -5741.22,E2 -5741.22} C_VEL
LIN {X 0,Y 502.065,Z 774.848,A -85,B 0,C 180,E1 -5743.743,E2 -5743.743} C_VEL
LIN {X 0,Y 502.09,Z 777.064,A -85,B 0,C 180,E1 -5745.796,E2 -5745.796} C_VEL
LIN {X 0,Y 504.472,Z 790.306,A -85,B 0,C 180,E1 -5746.25,E2 -5746.25} C_VEL
LIN {X 0,Y 504.263,Z 802.634,A -85,B 0,C 180,E1 -5746.757,E2 -5746.757} C_VEL
LIN {X 0,Y 503.997,Z 812.469,A -85,B 0,C 180,E1 -5747.284,E2 -5747.284} C_VEL
LIN {X 0,Y 503.76,Z 822.032,A -85,B 0,C 180,E1 -5747.922,E2 -5747.922} C_VEL
LIN {X 0,Y 503.472,Z 830.814,A -85,B 0,C 180,E1 -5748.629,E2 -5748.629} C_VEL
LIN {X 0,Y 503.192,Z 838.256,A -85,B 0,C 180,E1 -5749.336,E2 -5749.336} C_VEL
LIN {X 0,Y 502.974,Z 845.494,A -85,B 0,C 180,E1 -5750.145,E2 -5750.145} C_VEL
LIN {X 0,Y 502.715,Z 853.038,A -85,B 0,C 180,E1 -5751.155,E2 -5751.155} C_VEL
LIN {X 0,Y 502.471,Z 859.327,A -85,B 0,C 180,E1 -5752.163,E2 -5752.163} C_VEL
LIN {X 0,Y 502.32,Z 864.78,A -85,B 0,C 180,E1 -5753.211,E2 -5753.211} C_VEL
LIN {X 0,Y 502.26,Z 869.711,A -85,B 0,C 180,E1 -5754.38,E2 -5754.38} C_VEL
LIN {X 0,Y 502.127,Z 873.689,A -85,B 0,C 180,E1 -5755.586,E2 -5755.586} C_VEL
LIN {X 0,Y 502.121,Z 876.638,A -85,B 0,C 180,E1 -5756.791,E2 -5756.791} C_VEL
LIN {X 0,Y 502.065,Z 878.147,A -85,B 0,C 180,E1 -5757.594,E2 -5757.594} C_VEL
LIN {X 0,Y 501.991,Z 879.702,A -85,B 0,C 180,E1 -5759.199,E2 -5759.199} C_VEL
LIN {X 0,Y 501.98,Z 879.999,A -85,B 0,C 180,E1 -5760.001,E2 -5760.001} C_VEL
LIN {X 0,Y 502.036,Z 879.181,A -85,B 0,C 180,E1 -5761.605,E2 -5761.605} C_VEL
LIN {X 0,Y 502.065,Z 878.279,A -85,B 0,C 180,E1 -5762.408,E2 -5762.408} C_VEL
LIN {X 0,Y 502.152,Z 875.016,A -85,B 0,C 180,E1 -5764.014,E2 -5764.014} C_VEL
LIN {X 0,Y 502.185,Z 871.456,A -85,B 0,C 180,E1 -5765.22,E2 -5765.22} C_VEL
LIN {X 0,Y 502.276,Z 868.568,A -85,B 0,C 180,E1 -5766.025,E2 -5766.025} C_VEL
LIN {X 0,Y 502.35,Z 863.078,A -85,B 0,C 180,E1 -5767.234,E2 -5767.234} C_VEL
LIN {X 0,Y 502.574,Z 856.246,A -85,B 0,C 180,E1 -5768.444,E2 -5768.444} C_VEL
LIN {X 0,Y 502.791,Z 849.337,A -85,B 0,C 180,E1 -5769.454,E2 -5769.454} C_VEL
LIN {X 0,Y 503.01,Z 842.82,A -85,B 0,C 180,E1 -5770.262,E2 -5770.262} C_VEL
LIN {X 0,Y 503.356,Z 834.039,A -85,B 0,C 180,E1 -5771.171,E2 -5771.171} C_VEL
LIN {X 0,Y 503.695,Z 824.576,A -85,B 0,C 180,E1 -5771.98,E2 -5771.98} C_VEL
LIN {X 0,Y 503.939,Z 815.137,A -85,B 0,C 180,E1 -5772.643,E2 -5772.643} C_VEL
LIN {X 0,Y 504.291,Z 803.471,A -85,B 0,C 180,E1 -5773.295,E2 -5773.295} C_VEL
LIN {X 0,Y 504.553,Z 791.362,A -85,B 0,C 180,E1 -5773.801,E2 -5773.801} C_VEL
LIN {X 0,Y 502.323,Z 778.641,A -85,B 0,C 180,E1 -5774.236,E2 -5774.236} C_VEL
LIN {X 0,Y 502.092,Z 777.371,A -85,B 0,C 180,E1 -5774.283,E2 -5774.283} C_VEL
LIN {X 0,Y 502.15,Z 773.676,A -85,B 0,C 180,E1 -5777.877,E2 -5777.877} C_VEL
LIN {X 0,Y 502.158,Z 770.792,A -85,B 0,C 180,E1 -5780.481,E2 -5780.481} C_VEL
LIN {X 0,Y 502.188,Z 767.899,A -85,B 0,C 180,E1 -5783.071,E2 -5783.071} C_VEL
LIN {X 0,Y 502.202,Z 764.808,A -85,B 0,C 180,E1 -5785.711,E2 -5785.711} C_VEL
LIN {X 0,Y 502.196,Z 761.428,A -85,B 0,C 180,E1 -5788.413,E2 -5788.413} C_VEL
LIN {X 0,Y 502.16,Z 758.992,A -85,B 0,C 180,E1 -5790.255,E2 -5790.255} C_VEL
LIN {X 0,Y 502.517,Z 758.893,A -85,B 0,C 180,E1 -5793.055,E2 -5793.055} C_VEL
LIN {X 0,Y 502.748,Z 758.859,A -85,B 0,C 180,E1 -5795.826,E2 -5795.826} C_VEL
LIN {X 0,Y 502.806,Z 758.856,A -85,B 0,C 180,E1 -5798.976,E2 -5798.976} C_VEL
LIN {X 0,Y 502.808,Z 758.85,A -85,B 0,C 180,E1 -5802.199,E2 -5802.199} C_VEL
LIN {X 0,Y 502.806,Z 758.853,A -85,B 0,C 180,E1 -5805.468,E2 -5805.468} C_VEL
LIN {X 0,Y 502.824,Z 758.854,A -85,B 0,C 180,E1 -5808.934,E2 -5808.934} C_VEL
LIN {X 0,Y 502.828,Z 758.881,A -85,B 0,C 180,E1 -5810.639,E2 -5810.639} C_VEL
LIN {X 0,Y 504.092,Z 766.117,A -85,B 0,C 180,E1 -5813.6,E2 -5813.6} C_VEL
LIN {X 0,Y 504.212,Z 770.638,A -85,B 0,C 180,E1 -5815.324,E2 -5815.324} C_VEL
LIN {X 0,Y 503.856,Z 778.828,A -85,B 0,C 180,E1 -5818.306,E2 -5818.306} C_VEL
LIN {X 0,Y 503.521,Z 787.133,A -85,B 0,C 180,E1 -5821.21,E2 -5821.21} C_VEL
LIN {X 0,Y 503.269,Z 795.086,A -85,B 0,C 180,E1 -5823.903,E2 -5823.903} C_VEL
LIN {X 0,Y 503.032,Z 804.429,A -85,B 0,C 180,E1 -5826.971,E2 -5826.971} C_VEL
LIN {X 0,Y 502.786,Z 813.821,A -85,B 0,C 180,E1 -5829.973,E2 -5829.973} C_VEL
LIN {X 0,Y 502.6,Z 823.325,A -85,B 0,C 180,E1 -5832.923,E2 -5832.923} C_VEL
LIN {X 0,Y 502.476,Z 832.31,A -85,B 0,C 180,E1 -5835.677,E2 -5835.677} C_VEL
LIN {X 0,Y 504.682,Z 846.685,A -85,B 0,C 180,E1 -5836.101,E2 -5836.101} C_VEL
LIN {X 0,Y 504.382,Z 860.069,A -85,B 0,C 180,E1 -5836.606,E2 -5836.606} C_VEL
LIN {X 0,Y 504.019,Z 872.81,A -85,B 0,C 180,E1 -5837.267,E2 -5837.267} C_VEL
LIN {X 0,Y 503.689,Z 883.893,A -85,B 0,C 180,E1 -5838.021,E2 -5838.021} C_VEL
LIN {X 0,Y 503.337,Z 894.535,A -85,B 0,C 180,E1 -5838.931,E2 -5838.931} C_VEL
LIN {X 0,Y 503.007,Z 904.113,A -85,B 0,C 180,E1 -5839.942,E2 -5839.942} C_VEL
LIN {X 0,Y 502.705,Z 911.96,A -85,B 0,C 180,E1 -5840.951,E2 -5840.951} C_VEL
LIN {X 0,Y 502.471,Z 919.621,A -85,B 0,C 180,E1 -5842.162,E2 -5842.162} C_VEL
LIN {X 0,Y 502.257,Z 926.679,A -85,B 0,C 180,E1 -5843.573,E2 -5843.573} C_VEL
LIN {X 0,Y 502.186,Z 931.373,A -85,B 0,C 180,E1 -5844.781,E2 -5844.781} C_VEL
LIN {X 0,Y 502.152,Z 934.958,A -85,B 0,C 180,E1 -5845.987,E2 -5845.987} C_VEL
LIN {X 0,Y 502.121,Z 936.807,A -85,B 0,C 180,E1 -5846.791,E2 -5846.791} C_VEL
LIN {X 0,Y 502.036,Z 939.182,A -85,B 0,C 180,E1 -5848.396,E2 -5848.396} C_VEL
LIN {X 0,Y 501.98,Z 940,A -85,B 0,C 180,E1 -5850,E2 -5850} C_VEL
LIN {X 0,Y 502.036,Z 939.183,A -85,B 0,C 180,E1 -5851.604,E2 -5851.604} C_VEL
LIN {X 0,Y 502.121,Z 936.81,A -85,B 0,C 180,E1 -5853.209,E2 -5853.209} C_VEL
LIN {X 0,Y 502.129,Z 933.895,A -85,B 0,C 180,E1 -5854.415,E2 -5854.415} C_VEL
LIN {X 0,Y 502.26,Z 929.948,A -85,B 0,C 180,E1 -5855.621,E2 -5855.621} C_VEL
LIN {X 0,Y 502.337,Z 923.976,A -85,B 0,C 180,E1 -5857.012,E2 -5857.012} C_VEL
LIN {X 0,Y 502.543,Z 917.235,A -85,B 0,C 180,E1 -5858.241,E2 -5858.241} C_VEL
LIN {X 0,Y 502.812,Z 908.992,A -85,B 0,C 180,E1 -5859.453,E2 -5859.453} C_VEL
LIN {X 0,Y 503.06,Z 900.539,A -85,B 0,C 180,E1 -5860.464,E2 -5860.464} C_VEL
LIN {X 0,Y 503.538,Z 890.089,A -85,B 0,C 180,E1 -5861.472,E2 -5861.472} C_VEL
LIN {X 0,Y 503.824,Z 879.386,A -85,B 0,C 180,E1 -5862.306,E2 -5862.306} C_VEL
LIN {X 0,Y 504.136,Z 868.26,A -85,B 0,C 180,E1 -5862.991,E2 -5862.991} C_VEL
LIN {X 0,Y 504.467,Z 856.496,A -85,B 0,C 180,E1 -5863.546,E2 -5863.546} C_VEL
LIN {X 0,Y 504.581,Z 845.243,A -85,B 0,C 180,E1 -5863.941,E2 -5863.941} C_VEL
LIN {X 0,Y 502.476,Z 832.154,A -85,B 0,C 180,E1 -5864.323,E2 -5864.323} C_VEL
LIN {X 0,Y 502.611,Z 821.547,A -85,B 0,C 180,E1 -5867.496,E2 -5867.496} C_VEL
LIN {X 0,Y 502.771,Z 811.506,A -85,B 0,C 180,E1 -5870.517,E2 -5870.517} C_VEL
LIN {X 0,Y 502.96,Z 802.016,A -85,B 0,C 180,E1 -5873.468,E2 -5873.468} C_VEL
LIN {X 0,Y 503.142,Z 792.147,A -85,B 0,C 180,E1 -5876.623,E2 -5876.623} C_VEL
LIN {X 0,Y 503.331,Z 784.341,A -85,B 0,C 180,E1 -5879.256,E2 -5879.256} C_VEL
LIN {X 0,Y 503.671,Z 776.667,A -85,B 0,C 180,E1 -5882.022,E2 -5882.022} C_VEL
LIN {X 0,Y 504.097,Z 769.568,A -85,B 0,C 180,E1 -5884.863,E2 -5884.863} C_VEL
LIN {X 0,Y 504.138,Z 766.938,A -85,B 0,C 180,E1 -5886.044,E2 -5886.044} C_VEL
LIN {X 0,Y 503.595,Z 763.395,A -85,B 0,C 180,E1 -5887.883,E2 -5887.883} C_VEL
LIN {X 0,Y 502.893,Z 759.388,A -85,B 0,C 180,E1 -5890.53,E2 -5890.53} C_VEL
LIN {X 0,Y 502.824,Z 758.854,A -85,B 0,C 180,E1 -5891.066,E2 -5891.066} C_VEL
LIN {X 0,Y 502.806,Z 758.857,A -85,B 0,C 180,E1 -5894.532,E2 -5894.532} C_VEL
LIN {X 0,Y 502.799,Z 758.855,A -85,B 0,C 180,E1 -5897.86,E2 -5897.86} C_VEL
LIN {X 0,Y 502.803,Z 758.857,A -85,B 0,C 180,E1 -5901.023,E2 -5901.023} C_VEL
LIN {X 0,Y 502.75,Z 758.863,A -85,B 0,C 180,E1 -5904.173,E2 -5904.173} C_VEL
LIN {X 0,Y 502.702,Z 758.925,A -85,B 0,C 180,E1 -5905.026,E2 -5905.026} C_VEL
LIN {X 0,Y 502.693,Z 760.39,A -85,B 0,C 180,E1 -5907.018,E2 -5907.018} C_VEL
LIN {X 0,Y 502.537,Z 762.908,A -85,B 0,C 180,E1 -5910.121,E2 -5910.121} C_VEL
LIN {X 0,Y 502.403,Z 765.738,A -85,B 0,C 180,E1 -5913.407,E2 -5913.407} C_VEL
LIN {X 0,Y 502.305,Z 768.132,A -85,B 0,C 180,E1 -5916.061,E2 -5916.061} C_VEL
LIN {X 0,Y 502.263,Z 770.569,A -85,B 0,C 180,E1 -5918.665,E2 -5918.665} C_VEL
LIN {X 0,Y 502.165,Z 773.018,A -85,B 0,C 180,E1 -5921.222,E2 -5921.222} C_VEL
LIN {X 0,Y 502.104,Z 775.444,A -85,B 0,C 180,E1 -5923.743,E2 -5923.743} C_VEL
LIN {X 0,Y 502.124,Z 777.553,A -85,B 0,C 180,E1 -5925.821,E2 -5925.821} C_VEL
LIN {X 0,Y 504.499,Z 790.705,A -85,B 0,C 180,E1 -5926.262,E2 -5926.262} C_VEL
LIN {X 0,Y 504.33,Z 802.792,A -85,B 0,C 180,E1 -5926.757,E2 -5926.757} C_VEL
LIN {X 0,Y 504.011,Z 814.568,A -85,B 0,C 180,E1 -5927.405,E2 -5927.405} C_VEL
LIN {X 0,Y 503.658,Z 826.104,A -85,B 0,C 180,E1 -5928.224,E2 -5928.224} C_VEL
LIN {X 0,Y 503.277,Z 836.356,A -85,B 0,C 180,E1 -5929.133,E2 -5929.133} C_VEL
LIN {X 0,Y 502.968,Z 845.546,A -85,B 0,C 180,E1 -5930.143,E2 -5930.143} C_VEL
LIN {X 0,Y 502.637,Z 854.445,A -85,B 0,C 180,E1 -5931.354,E2 -5931.354} C_VEL
LIN {X 0,Y 502.374,Z 861.601,A -85,B 0,C 180,E1 -5932.564,E2 -5932.564} C_VEL
LIN {X 0,Y 502.276,Z 866.473,A -85,B 0,C 180,E1 -5933.572,E2 -5933.572} C_VEL
LIN {X 0,Y 502.186,Z 871.21,A -85,B 0,C 180,E1 -5934.78,E2 -5934.78} C_VEL
LIN {X 0,Y 502.152,Z 874.839,A -85,B 0,C 180,E1 -5935.986,E2 -5935.986} C_VEL
LIN {X 0,Y 502.122,Z 876.715,A -85,B 0,C 180,E1 -5936.79,E2 -5936.79} C_VEL
LIN {X 0,Y 502.066,Z 878.131,A -85,B 0,C 180,E1 -5937.592,E2 -5937.592} C_VEL
LIN {X 0,Y 501.991,Z 879.758,A -85,B 0,C 180,E1 -5939.197,E2 -5939.197} C_VEL
LIN {X 0,Y 501.98,Z 879.997,A -85,B 0,C 180,E1 -5939.999,E2 -5939.999} C_VEL
LIN {X 0,Y 501.99,Z 879.813,A -85,B 0,C 180,E1 -5940.801,E2 -5940.801} C_VEL
LIN {X 0,Y 502.065,Z 878.257,A -85,B 0,C 180,E1 -5942.406,E2 -5942.406} C_VEL
LIN {X 0,Y 502.121,Z 876.895,A -85,B 0,C 180,E1 -5943.209,E2 -5943.209} C_VEL
LIN {X 0,Y 502.128,Z 874.016,A -85,B 0,C 180,E1 -5944.414,E2 -5944.414} C_VEL
LIN {X 0,Y 502.25,Z 870.112,A -85,B 0,C 180,E1 -5945.62,E2 -5945.62} C_VEL
LIN {X 0,Y 502.308,Z 865.078,A -85,B 0,C 180,E1 -5946.829,E2 -5946.829} C_VEL
LIN {X 0,Y 502.504,Z 858.759,A -85,B 0,C 180,E1 -5948.039,E2 -5948.039} C_VEL
LIN {X 0,Y 502.762,Z 850.882,A -85,B 0,C 180,E1 -5949.25,E2 -5949.25} C_VEL
LIN {X 0,Y 503.062,Z 841.07,A -85,B 0,C 180,E1 -5950.463,E2 -5950.463} C_VEL
LIN {X 0,Y 503.486,Z 830.758,A -85,B 0,C 180,E1 -5951.472,E2 -5951.472} C_VEL
LIN {X 0,Y 503.756,Z 820.311,A -85,B 0,C 180,E1 -5952.299,E2 -5952.299} C_VEL
LIN {X 0,Y 504.118,Z 809.351,A -85,B 0,C 180,E1 -5952.99,E2 -5952.99} C_VEL
LIN {X 0,Y 504.451,Z 798.011,A -85,B 0,C 180,E1 -5953.545,E2 -5953.545} C_VEL
LIN {X 0,Y 504.4,Z 789.926,A -85,B 0,C 180,E1 -5953.855,E2 -5953.855} C_VEL
LIN {X 0,Y 502.087,Z 777.122,A -85,B 0,C 180,E1 -5954.282,E2 -5954.282} C_VEL
LIN {X 0,Y 502.083,Z 774.067,A -85,B 0,C 180,E1 -5957.094,E2 -5957.094} C_VEL
LIN {X 0,Y 502.152,Z 770.518,A -85,B 0,C 180,E1 -5960.48,E2 -5960.48} C_VEL
LIN {X 0,Y 502.195,Z 767.754,A -85,B 0,C 180,E1 -5963.068,E2 -5963.068} C_VEL
LIN {X 0,Y 502.21,Z 764.919,A -85,B 0,C 180,E1 -5965.709,E2 -5965.709} C_VEL
LIN {X 0,Y 502.253,Z 762.117,A -85,B 0,C 180,E1 -5968.408,E2 -5968.408} C_VEL
LIN {X 0,Y 502.324,Z 759.228,A -85,B 0,C 180,E1 -5971.175,E2 -5971.175} C_VEL
LIN {X 0,Y 502.482,Z 758.896,A -85,B 0,C 180,E1 -5973.056,E2 -5973.056} C_VEL
LIN {X 0,Y 502.687,Z 758.871,A -85,B 0,C 180,E1 -5974.973,E2 -5974.973} C_VEL
LIN {X 0,Y 502.786,Z 758.853,A -85,B 0,C 180,E1 -5977.953,E2 -5977.953} C_VEL
LIN {X 0,Y 502.815,Z 758.854,A -85,B 0,C 180,E1 -5981.065,E2 -5981.065} C_VEL
LIN {X 0,Y 502.795,Z 758.851,A -85,B 0,C 180,E1 -5984.531,E2 -5984.531} C_VEL
LIN {X 0,Y 502.789,Z 758.854,A -85,B 0,C 180,E1 -5987.86,E2 -5987.86} C_VEL
LIN {X 0,Y 502.794,Z 758.854,A -85,B 0,C 180,E1 -5991.023,E2 -5991.023} C_VEL
LIN {X 0,Y 502.755,Z 758.857,A -85,B 0,C 180,E1 -5993.23,E2 -5993.23} C_VEL
LIN {X 0,Y 502.088,Z 758.942,A -85,B 0,C 180,E1 -5993.899,E2 -5993.899} C_VEL
LIN {X 0,Y 499.29,Z 759.29,A -85,B 0,C 180,E1 -5994.986,E2 -5994.986} C_VEL
LIN {X 0,Y 496.917,Z 759.587,A -85,B 0,C 180,E1 -5995.862,E2 -5995.862} C_VEL
LIN {X 0,Y 495.877,Z 759.713,A -85,B 0,C 180,E1 -5996.537,E2 -5996.537} C_VEL
LIN {X 0,Y 495.781,Z 759.725,A -85,B 0,C 180,E1 -5996.766,E2 -5996.766} C_VEL
LIN {X 0,Y 495.756,Z 759.732,A -85,B 0,C 180,E1 -5999.852,E2 -5999.852} C_VEL
LIN {X 0,Y 495.752,Z 759.729,A -85,B 0,C 180,E1 -6003.022,E2 -6003.022} C_VEL
LIN {X 0,Y 495.707,Z 759.739,A -85,B 0,C 180,E1 -6005.723,E2 -6005.723} C_VEL
LIN {X 0,Y 495.733,Z 759.731,A -85,B 0,C 180,E1 -6008.37,E2 -6008.37} C_VEL
LIN {X 0,Y 495.769,Z 759.726,A -85,B 0,C 180,E1 -6010.971,E2 -6010.971} C_VEL
LIN {X 0,Y 495.814,Z 759.72,A -85,B 0,C 180,E1 -6014.548,E2 -6014.548} C_VEL
LIN {X 0,Y 495.819,Z 759.725,A -85,B 0,C 180,E1 -6017.965,E2 -6017.965} C_VEL
LIN {X 0,Y 495.795,Z 759.722,A -85,B 0,C 180,E1 -6021.029,E2 -6021.029} C_VEL
LIN {X 0,Y 495.809,Z 759.723,A -85,B 0,C 180,E1 -6023.489,E2 -6023.489} C_VEL
LIN {X 0,Y 495.693,Z 759.743,A -85,B 0,C 180,E1 -6025.935,E2 -6025.935} C_VEL
LIN {X 0,Y 495.964,Z 759.703,A -85,B 0,C 180,E1 -6027.564,E2 -6027.564} C_VEL
LIN {X 0,Y 495.961,Z 759.709,A -85,B 0,C 180,E1 -6030,E2 -6030} C_VEL
LIN {X 0,Y 495.962,Z 759.704,A -85,B 0,C 180,E1 -6032.436,E2 -6032.436} C_VEL
LIN {X 0,Y 495.838,Z 759.719,A -85,B 0,C 180,E1 -6035.694,E2 -6035.694} C_VEL
LIN {X 0,Y 495.799,Z 759.73,A -85,B 0,C 180,E1 -6038.149,E2 -6038.149} C_VEL
LIN {X 0,Y 495.81,Z 759.72,A -85,B 0,C 180,E1 -6041.446,E2 -6041.446} C_VEL
LIN {X 0,Y 495.777,Z 759.726,A -85,B 0,C 180,E1 -6044.783,E2 -6044.783} C_VEL
LIN {X 0,Y 495.769,Z 759.731,A -85,B 0,C 180,E1 -6048.172,E2 -6048.172} C_VEL
LIN {X 0,Y 495.765,Z 759.729,A -85,B 0,C 180,E1 -6050.757,E2 -6050.757} C_VEL
LIN {X 0,Y 495.73,Z 759.73,A -85,B 0,C 180,E1 -6053.388,E2 -6053.388} C_VEL
LIN {X 0,Y 495.733,Z 759.735,A -85,B 0,C 180,E1 -6056.731,E2 -6056.731} C_VEL
LIN {X 0,Y 495.754,Z 759.728,A -85,B 0,C 180,E1 -6059.747,E2 -6059.747} C_VEL
LIN {X 0,Y 495.758,Z 759.734,A -85,B 0,C 180,E1 -6062.595,E2 -6062.595} C_VEL
LIN {X 0,Y 495.739,Z 759.73,A -85,B 0,C 180,E1 -6065.539,E2 -6065.539} C_VEL
LIN {X 0,Y 495.756,Z 759.735,A -85,B 0,C 180,E1 -6068.769,E2 -6068.769} C_VEL
LIN {X 0,Y 495.75,Z 759.729,A -85,B 0,C 180,E1 -6071.782,E2 -6071.782} C_VEL
LIN {X 0,Y 495.732,Z 759.734,A -85,B 0,C 180,E1 -6075.142,E2 -6075.142} C_VEL
LIN {X 0,Y 495.751,Z 759.73,A -85,B 0,C 180,E1 -6078.22,E2 -6078.22} C_VEL
LIN {X 0,Y 495.746,Z 759.731,A -85,B 0,C 180,E1 -6081.409,E2 -6081.409} C_VEL
LIN {X 0,Y 495.677,Z 759.741,A -85,B 0,C 180,E1 -6084.458,E2 -6084.458} C_VEL
LIN {X 0,Y 495.461,Z 759.772,A -85,B 0,C 180,E1 -6087.384,E2 -6087.384} C_VEL
LIN {X 0,Y 495.218,Z 759.802,A -85,B 0,C 180,E1 -6089.277,E2 -6089.277} C_VEL
LIN {X 0,Y 495.149,Z 760.508,A -85,B 0,C 180,E1 -6090.214,E2 -6090.214} C_VEL
LIN {X 0,Y 495.204,Z 764.1,A -85,B 0,C 180,E1 -6093.394,E2 -6093.394} C_VEL
LIN {X 0,Y 495.08,Z 767.613,A -85,B 0,C 180,E1 -6096.58,E2 -6096.58} C_VEL
LIN {X 0,Y 495.082,Z 770.844,A -85,B 0,C 180,E1 -6099.54,E2 -6099.54} C_VEL
LIN {X 0,Y 495.02,Z 774.207,A -85,B 0,C 180,E1 -6102.655,E2 -6102.655} C_VEL
LIN {X 0,Y 495.013,Z 777.465,A -85,B 0,C 180,E1 -6105.615,E2 -6105.615} C_VEL
LIN {X 0,Y 497.348,Z 790.046,A -85,B 0,C 180,E1 -6106.036,E2 -6106.036} C_VEL
LIN {X 0,Y 497.618,Z 794.536,A -85,B 0,C 180,E1 -6106.213,E2 -6106.213} C_VEL
LIN {X 0,Y 497.276,Z 805.89,A -85,B 0,C 180,E1 -6106.724,E2 -6106.724} C_VEL
LIN {X 0,Y 496.906,Z 817.911,A -85,B 0,C 180,E1 -6107.438,E2 -6107.438} C_VEL
LIN {X 0,Y 496.55,Z 829.939,A -85,B 0,C 180,E1 -6108.365,E2 -6108.365} C_VEL
LIN {X 0,Y 496.21,Z 838.528,A -85,B 0,C 180,E1 -6109.184,E2 -6109.184} C_VEL
LIN {X 0,Y 495.904,Z 847.379,A -85,B 0,C 180,E1 -6110.209,E2 -6110.209} C_VEL
LIN {X 0,Y 495.614,Z 854.689,A -85,B 0,C 180,E1 -6111.233,E2 -6111.233} C_VEL
LIN {X 0,Y 495.387,Z 860.777,A -85,B 0,C 180,E1 -6112.255,E2 -6112.255} C_VEL
LIN {X 0,Y 495.21,Z 866.734,A -85,B 0,C 180,E1 -6113.482,E2 -6113.482} C_VEL
LIN {X 0,Y 495.123,Z 871.444,A -85,B 0,C 180,E1 -6114.707,E2 -6114.707} C_VEL
LIN {X 0,Y 495.071,Z 875.048,A -85,B 0,C 180,E1 -6115.931,E2 -6115.931} C_VEL
LIN {X 0,Y 494.974,Z 878.354,A -85,B 0,C 180,E1 -6117.56,E2 -6117.56} C_VEL
LIN {X 0,Y 494.911,Z 879.92,A -85,B 0,C 180,E1 -6119.187,E2 -6119.187} C_VEL
LIN {X 0,Y 494.898,Z 880.197,A -85,B 0,C 180,E1 -6120.001,E2 -6120.001} C_VEL
LIN {X 0,Y 494.961,Z 879.407,A -85,B 0,C 180,E1 -6121.628,E2 -6121.628} C_VEL
LIN {X 0,Y 494.974,Z 878.494,A -85,B 0,C 180,E1 -6122.442,E2 -6122.442} C_VEL
LIN {X 0,Y 495.072,Z 875.295,A -85,B 0,C 180,E1 -6124.071,E2 -6124.071} C_VEL
LIN {X 0,Y 495.122,Z 871.777,A -85,B 0,C 180,E1 -6125.295,E2 -6125.295} C_VEL
LIN {X 0,Y 495.205,Z 867.162,A -85,B 0,C 180,E1 -6126.52,E2 -6126.52} C_VEL
LIN {X 0,Y 495.387,Z 861.317,A -85,B 0,C 180,E1 -6127.746,E2 -6127.746} C_VEL
LIN {X 0,Y 495.65,Z 854.036,A -85,B 0,C 180,E1 -6128.974,E2 -6128.974} C_VEL
LIN {X 0,Y 495.988,Z 844.913,A -85,B 0,C 180,E1 -6130.203,E2 -6130.203} C_VEL
LIN {X 0,Y 496.405,Z 834.383,A -85,B 0,C 180,E1 -6131.33,E2 -6131.33} C_VEL
LIN {X 0,Y 496.787,Z 823.548,A -85,B 0,C 180,E1 -6132.252,E2 -6132.252} C_VEL
LIN {X 0,Y 497.135,Z 812.808,A -85,B 0,C 180,E1 -6132.982,E2 -6132.982} C_VEL
LIN {X 0,Y 497.495,Z 800.41,A -85,B 0,C 180,E1 -6133.636,E2 -6133.636} C_VEL
LIN {X 0,Y 497.538,Z 791.431,A -85,B 0,C 180,E1 -6133.999,E2 -6133.999} C_VEL
LIN {X 0,Y 495.441,Z 779.692,A -85,B 0,C 180,E1 -6134.414,E2 -6134.414} C_VEL
LIN {X 0,Y 495.039,Z 777.888,A -85,B 0,C 180,E1 -6134.491,E2 -6134.491} C_VEL
LIN {X 0,Y 495.073,Z 774.193,A -85,B 0,C 180,E1 -6137.987,E2 -6137.987} C_VEL
LIN {X 0,Y 495.086,Z 771.106,A -85,B 0,C 180,E1 -6140.787,E2 -6140.787} C_VEL
LIN {X 0,Y 495.129,Z 768.23,A -85,B 0,C 180,E1 -6143.419,E2 -6143.419} C_VEL
LIN {X 0,Y 495.144,Z 764.403,A -85,B 0,C 180,E1 -6146.592,E2 -6146.592} C_VEL
LIN {X 0,Y 495.111,Z 761.497,A -85,B 0,C 180,E1 -6148.858,E2 -6148.858} C_VEL
LIN {X 0,Y 495.098,Z 759.957,A -85,B 0,C 180,E1 -6150.013,E2 -6150.013} C_VEL
LIN {X 0,Y 495.433,Z 759.775,A -85,B 0,C 180,E1 -6152.62,E2 -6152.62} C_VEL
LIN {X 0,Y 495.678,Z 759.742,A -85,B 0,C 180,E1 -6155.544,E2 -6155.544} C_VEL
LIN {X 0,Y 495.768,Z 759.731,A -85,B 0,C 180,E1 -6158.768,E2 -6158.768} C_VEL
LIN {X 0,Y 495.755,Z 759.729,A -85,B 0,C 180,E1 -6161.782,E2 -6161.782} C_VEL
LIN {X 0,Y 495.754,Z 759.735,A -85,B 0,C 180,E1 -6165.14,E2 -6165.14} C_VEL
LIN {X 0,Y 495.761,Z 759.729,A -85,B 0,C 180,E1 -6168.219,E2 -6168.219} C_VEL
LIN {X 0,Y 495.764,Z 759.767,A -85,B 0,C 180,E1 -6170.363,E2 -6170.363} C_VEL
LIN {X 0,Y 496.94,Z 766.213,A -85,B 0,C 180,E1 -6173.054,E2 -6173.054} C_VEL
LIN {X 0,Y 497.303,Z 770.096,A -85,B 0,C 180,E1 -6174.59,E2 -6174.59} C_VEL
LIN {X 0,Y 496.95,Z 777.858,A -85,B 0,C 180,E1 -6177.493,E2 -6177.493} C_VEL
LIN {X 0,Y 496.565,Z 787.022,A -85,B 0,C 180,E1 -6180.772,E2 -6180.772} C_VEL
LIN {X 0,Y 496.252,Z 796.239,A -85,B 0,C 180,E1 -6183.958,E2 -6183.958} C_VEL
LIN {X 0,Y 495.989,Z 804.214,A -85,B 0,C 180,E1 -6186.625,E2 -6186.625} C_VEL
LIN {X 0,Y 495.765,Z 813.697,A -85,B 0,C 180,E1 -6189.716,E2 -6189.716} C_VEL
LIN {X 0,Y 495.543,Z 822.995,A -85,B 0,C 180,E1 -6192.673,E2 -6192.673} C_VEL
LIN {X 0,Y 495.408,Z 832.029,A -85,B 0,C 180,E1 -6195.494,E2 -6195.494} C_VEL
LIN {X 0,Y 497.59,Z 845.661,A -85,B 0,C 180,E1 -6195.885,E2 -6195.885} C_VEL
LIN {X 0,Y 497.487,Z 858.373,A -85,B 0,C 180,E1 -6196.364,E2 -6196.364} C_VEL
LIN {X 0,Y 497.063,Z 871.003,A -85,B 0,C 180,E1 -6197.012,E2 -6197.012} C_VEL
LIN {X 0,Y 496.734,Z 882.046,A -85,B 0,C 180,E1 -6197.747,E2 -6197.747} C_VEL
LIN {X 0,Y 496.38,Z 893.046,A -85,B 0,C 180,E1 -6198.671,E2 -6198.671} C_VEL
LIN {X 0,Y 495.996,Z 902.006,A -85,B 0,C 180,E1 -6199.592,E2 -6199.592} C_VEL
LIN {X 0,Y 495.674,Z 911.747,A -85,B 0,C 180,E1 -6200.821,E2 -6200.821} C_VEL
LIN {X 0,Y 495.401,Z 919.502,A -85,B 0,C 180,E1 -6202.049,E2 -6202.049} C_VEL
LIN {X 0,Y 495.185,Z 926.648,A -85,B 0,C 180,E1 -6203.48,E2 -6203.48} C_VEL
LIN {X 0,Y 495.123,Z 931.372,A -85,B 0,C 180,E1 -6204.706,E2 -6204.706} C_VEL
LIN {X 0,Y 495.05,Z 934.957,A -85,B 0,C 180,E1 -6205.93,E2 -6205.93} C_VEL
LIN {X 0,Y 495.044,Z 936.806,A -85,B 0,C 180,E1 -6206.745,E2 -6206.745} C_VEL
LIN {X 0,Y 494.961,Z 939.181,A -85,B 0,C 180,E1 -6208.373,E2 -6208.373} C_VEL
LIN {X 0,Y 494.898,Z 940,A -85,B 0,C 180,E1 -6210,E2 -6210} C_VEL
LIN {X 0,Y 494.961,Z 939.183,A -85,B 0,C 180,E1 -6211.627,E2 -6211.627} C_VEL
LIN {X 0,Y 495.044,Z 936.81,A -85,B 0,C 180,E1 -6213.255,E2 -6213.255} C_VEL
LIN {X 0,Y 495.029,Z 933.895,A -85,B 0,C 180,E1 -6214.478,E2 -6214.478} C_VEL
LIN {X 0,Y 495.179,Z 929.944,A -85,B 0,C 180,E1 -6215.702,E2 -6215.702} C_VEL
LIN {X 0,Y 495.252,Z 923.908,A -85,B 0,C 180,E1 -6217.112,E2 -6217.112} C_VEL
LIN {X 0,Y 495.486,Z 917.067,A -85,B 0,C 180,E1 -6218.36,E2 -6218.36} C_VEL
LIN {X 0,Y 495.771,Z 908.699,A -85,B 0,C 180,E1 -6219.588,E2 -6219.588} C_VEL
LIN {X 0,Y 496.058,Z 900.107,A -85,B 0,C 180,E1 -6220.613,E2 -6220.613} C_VEL
LIN {X 0,Y 496.53,Z 889.503,A -85,B 0,C 180,E1 -6221.636,E2 -6221.636} C_VEL
LIN {X 0,Y 496.826,Z 877.563,A -85,B 0,C 180,E1 -6222.561,E2 -6222.561} C_VEL
LIN {X 0,Y 497.198,Z 865.518,A -85,B 0,C 180,E1 -6223.279,E2 -6223.279} C_VEL
LIN {X 0,Y 497.602,Z 853.039,A -85,B 0,C 180,E1 -6223.841,E2 -6223.841} C_VEL
LIN {X 0,Y 497.543,Z 845.7,A -85,B 0,C 180,E1 -6224.103,E2 -6224.103} C_VEL
LIN {X 0,Y 495.389,Z 831.72,A -85,B 0,C 180,E1 -6224.506,E2 -6224.506} C_VEL
LIN {X 0,Y 495.547,Z 821.062,A -85,B 0,C 180,E1 -6227.747,E2 -6227.747} C_VEL
LIN {X 0,Y 495.7,Z 811.215,A -85,B 0,C 180,E1 -6230.76,E2 -6230.76} C_VEL
LIN {X 0,Y 495.901,Z 801.584,A -85,B 0,C 180,E1 -6233.823,E2 -6233.823} C_VEL
LIN {X 0,Y 496.134,Z 792.42,A -85,B 0,C 180,E1 -6236.819,E2 -6236.819} C_VEL
LIN {X 0,Y 496.37,Z 784.119,A -85,B 0,C 180,E1 -6239.707,E2 -6239.707} C_VEL
LIN {X 0,Y 496.762,Z 776.584,A -85,B 0,C 180,E1 -6242.521,E2 -6242.521} C_VEL
LIN {X 0,Y 497.171,Z 769.7,A -85,B 0,C 180,E1 -6245.421,E2 -6245.421} C_VEL
LIN {X 0,Y 497.102,Z 767.601,A -85,B 0,C 180,E1 -6246.427,E2 -6246.427} C_VEL
LIN {X 0,Y 496.385,Z 763.314,A -85,B 0,C 180,E1 -6248.857,E2 -6248.857} C_VEL
LIN {X 0,Y 495.836,Z 760.061,A -85,B 0,C 180,E1 -6251.303,E2 -6251.303} C_VEL
LIN {X 0,Y 495.743,Z 759.735,A -85,B 0,C 180,E1 -6252.507,E2 -6252.507} C_VEL
LIN {X 0,Y 495.754,Z 759.735,A -85,B 0,C 180,E1 -6255.139,E2 -6255.139} C_VEL
LIN {X 0,Y 495.754,Z 759.733,A -85,B 0,C 180,E1 -6258.218,E2 -6258.218} C_VEL
LIN {X 0,Y 495.753,Z 759.735,A -85,B 0,C 180,E1 -6261.408,E2 -6261.408} C_VEL
LIN {X 0,Y 495.681,Z 759.745,A -85,B 0,C 180,E1 -6264.456,E2 -6264.456} C_VEL
LIN {X 0,Y 495.696,Z 761.249,A -85,B 0,C 180,E1 -6266.773,E2 -6266.773} C_VEL
LIN {X 0,Y 495.497,Z 763.685,A -85,B 0,C 180,E1 -6269.907,E2 -6269.907} C_VEL
LIN {X 0,Y 495.359,Z 766.276,A -85,B 0,C 180,E1 -6272.998,E2 -6272.998} C_VEL
LIN {X 0,Y 495.286,Z 768.64,A -85,B 0,C 180,E1 -6275.7,E2 -6275.7} C_VEL
LIN {X 0,Y 495.233,Z 771.07,A -85,B 0,C 180,E1 -6278.347,E2 -6278.347} C_VEL
LIN {X 0,Y 495.125,Z 773.534,A -85,B 0,C 180,E1 -6280.945,E2 -6280.945} C_VEL
LIN {X 0,Y 495.051,Z 775.971,A -85,B 0,C 180,E1 -6283.504,E2 -6283.504} C_VEL
LIN {X 0,Y 495.043,Z 778.076,A -85,B 0,C 180,E1 -6285.614,E2 -6285.614} C_VEL
LIN {X 0,Y 497.177,Z 789.013,A -85,B 0,C 180,E1 -6285.99,E2 -6285.99} C_VEL
LIN {X 0,Y 497.656,Z 793.417,A -85,B 0,C 180,E1 -6286.16,E2 -6286.16} C_VEL
LIN {X 0,Y 497.341,Z 806.054,A -85,B 0,C 180,E1 -6286.724,E2 -6286.724} C_VEL
LIN {X 0,Y 496.976,Z 818.485,A -85,B 0,C 180,E1 -6287.465,E2 -6287.465} C_VEL
LIN {X 0,Y 496.647,Z 828.902,A -85,B 0,C 180,E1 -6288.262,E2 -6288.262} C_VEL
LIN {X 0,Y 496.244,Z 838.659,A -85,B 0,C 180,E1 -6289.183,E2 -6289.183} C_VEL
LIN {X 0,Y 495.902,Z 847.522,A -85,B 0,C 180,E1 -6290.208,E2 -6290.208} C_VEL
LIN {X 0,Y 495.576,Z 856.162,A -85,B 0,C 180,E1 -6291.436,E2 -6291.436} C_VEL
LIN {X 0,Y 495.308,Z 863.038,A -85,B 0,C 180,E1 -6292.662,E2 -6292.662} C_VEL
LIN {X 0,Y 495.231,Z 868.959,A -85,B 0,C 180,E1 -6294.001,E2 -6294.001} C_VEL
LIN {X 0,Y 495.056,Z 874.057,A -85,B 0,C 180,E1 -6295.521,E2 -6295.521} C_VEL
LIN {X 0,Y 495.044,Z 876.964,A -85,B 0,C 180,E1 -6296.744,E2 -6296.744} C_VEL
LIN {X 0,Y 494.975,Z 878.365,A -85,B 0,C 180,E1 -6297.558,E2 -6297.558} C_VEL
LIN {X 0,Y 494.911,Z 879.97,A -85,B 0,C 180,E1 -6299.186,E2 -6299.186} C_VEL
LIN {X 0,Y 494.898,Z 880.203,A -85,B 0,C 180,E1 -6299.999,E2 -6299.999} C_VEL
LIN {X 0,Y 494.911,Z 880.018,A -85,B 0,C 180,E1 -6300.813,E2 -6300.813} C_VEL
LIN {X 0,Y 494.974,Z 878.474,A -85,B 0,C 180,E1 -6302.44,E2 -6302.44} C_VEL
LIN {X 0,Y 495.043,Z 877.12,A -85,B 0,C 180,E1 -6303.255,E2 -6303.255} C_VEL
LIN {X 0,Y 495.054,Z 874.269,A -85,B 0,C 180,E1 -6304.477,E2 -6304.477} C_VEL
LIN {X 0,Y 495.215,Z 869.311,A -85,B 0,C 180,E1 -6305.989,E2 -6305.989} C_VEL
LIN {X 0,Y 495.304,Z 863.423,A -85,B 0,C 180,E1 -6307.336,E2 -6307.336} C_VEL
LIN {X 0,Y 495.555,Z 856.636,A -85,B 0,C 180,E1 -6308.563,E2 -6308.563} C_VEL
LIN {X 0,Y 495.872,Z 848.145,A -85,B 0,C 180,E1 -6309.791,E2 -6309.791} C_VEL
LIN {X 0,Y 496.204,Z 839.41,A -85,B 0,C 180,E1 -6310.816,E2 -6310.816} C_VEL
LIN {X 0,Y 496.629,Z 828.644,A -85,B 0,C 180,E1 -6311.84,E2 -6311.84} C_VEL
LIN {X 0,Y 496.945,Z 817.548,A -85,B 0,C 180,E1 -6312.679,E2 -6312.679} C_VEL
LIN {X 0,Y 497.297,Z 805.68,A -85,B 0,C 180,E1 -6313.38,E2 -6313.38} C_VEL
LIN {X 0,Y 497.644,Z 792.999,A -85,B 0,C 180,E1 -6313.943,E2 -6313.943} C_VEL
LIN {X 0,Y 495.756,Z 781.047,A -85,B 0,C 180,E1 -6314.373,E2 -6314.373} C_VEL
LIN {X 0,Y 495.025,Z 777.489,A -85,B 0,C 180,E1 -6314.49,E2 -6314.49} C_VEL
LIN {X 0,Y 495.021,Z 774.4,A -85,B 0,C 180,E1 -6317.345,E2 -6317.345} C_VEL
LIN {X 0,Y 495.077,Z 770.767,A -85,B 0,C 180,E1 -6320.786,E2 -6320.786} C_VEL
LIN {X 0,Y 495.14,Z 767.96,A -85,B 0,C 180,E1 -6323.417,E2 -6323.417} C_VEL
LIN {X 0,Y 495.2,Z 764.577,A -85,B 0,C 180,E1 -6326.605,E2 -6326.605} C_VEL
LIN {X 0,Y 495.259,Z 761.04,A -85,B 0,C 180,E1 -6330.046,E2 -6330.046} C_VEL
LIN {X 0,Y 495.309,Z 759.791,A -85,B 0,C 180,E1 -6331.667,E2 -6331.667} C_VEL
LIN {X 0,Y 495.656,Z 759.747,A -85,B 0,C 180,E1 -6334.675,E2 -6334.675} C_VEL
LIN {X 0,Y 495.717,Z 759.737,A -85,B 0,C 180,E1 -6337.561,E2 -6337.561} C_VEL
LIN {X 0,Y 495.754,Z 759.729,A -85,B 0,C 180,E1 -6340.046,E2 -6340.046} C_VEL
LIN {X 0,Y 495.721,Z 759.736,A -85,B 0,C 180,E1 -6342.882,E2 -6342.882} C_VEL
LIN {X 0,Y 495.729,Z 759.733,A -85,B 0,C 180,E1 -6345.998,E2 -6345.998} C_VEL
LIN {X 0,Y 495.76,Z 759.734,A -85,B 0,C 180,E1 -6349.299,E2 -6349.299} C_VEL
LIN {X 0,Y 495.722,Z 759.732,A -85,B 0,C 180,E1 -6352.437,E2 -6352.437} C_VEL
LIN {X 0,Y 495.763,Z 759.733,A -85,B 0,C 180,E1 -6355.455,E2 -6355.455} C_VEL
LIN {X 0,Y 495.781,Z 759.725,A -85,B 0,C 180,E1 -6356.766,E2 -6356.766} C_VEL
LIN {X 0,Y 495.078,Z 759.819,A -85,B 0,C 180,E1 -6357.444,E2 -6357.444} C_VEL
LIN {X 0,Y 492.204,Z 760.174,A -85,B 0,C 180,E1 -6358.544,E2 -6358.544} C_VEL
LIN {X 0,Y 489.797,Z 760.477,A -85,B 0,C 180,E1 -6359.43,E2 -6359.43} C_VEL
LIN {X 0,Y 488.772,Z 760.6,A -85,B 0,C 180,E1 -6360.115,E2 -6360.115} C_VEL
LIN {X 0,Y 488.691,Z 760.607,A -85,B 0,C 180,E1 -6360.347,E2 -6360.347} C_VEL
LIN {X 0,Y 488.707,Z 760.613,A -85,B 0,C 180,E1 -6363.525,E2 -6363.525} C_VEL
LIN {X 0,Y 488.662,Z 760.613,A -85,B 0,C 180,E1 -6366.253,E2 -6366.253} C_VEL
LIN {X 0,Y 488.737,Z 760.604,A -85,B 0,C 180,E1 -6369.175,E2 -6369.175} C_VEL
LIN {X 0,Y 488.738,Z 760.609,A -85,B 0,C 180,E1 -6371.632,E2 -6371.632} C_VEL
LIN {X 0,Y 488.751,Z 760.6,A -85,B 0,C 180,E1 -6374.999,E2 -6374.999} C_VEL
LIN {X 0,Y 488.795,Z 760.596,A -85,B 0,C 180,E1 -6378.387,E2 -6378.387} C_VEL
LIN {X 0,Y 488.75,Z 760.606,A -85,B 0,C 180,E1 -6381.732,E2 -6381.732} C_VEL
LIN {X 0,Y 488.801,Z 760.597,A -85,B 0,C 180,E1 -6384.224,E2 -6384.224} C_VEL
LIN {X 0,Y 488.93,Z 760.579,A -85,B 0,C 180,E1 -6387.528,E2 -6387.528} C_VEL
LIN {X 0,Y 488.93,Z 760.585,A -85,B 0,C 180,E1 -6390,E2 -6390} C_VEL
LIN {X 0,Y 488.928,Z 760.58,A -85,B 0,C 180,E1 -6392.472,E2 -6392.472} C_VEL
LIN {X 0,Y 488.799,Z 760.596,A -85,B 0,C 180,E1 -6395.776,E2 -6395.776} C_VEL
LIN {X 0,Y 488.743,Z 760.608,A -85,B 0,C 180,E1 -6398.268,E2 -6398.268} C_VEL
LIN {X 0,Y 488.772,Z 760.598,A -85,B 0,C 180,E1 -6401.613,E2 -6401.613} C_VEL
LIN {X 0,Y 488.75,Z 760.6,A -85,B 0,C 180,E1 -6405.001,E2 -6405.001} C_VEL
LIN {X 0,Y 488.734,Z 760.609,A -85,B 0,C 180,E1 -6408.443,E2 -6408.443} C_VEL
LIN {X 0,Y 488.698,Z 760.607,A -85,B 0,C 180,E1 -6411.071,E2 -6411.071} C_VEL
LIN {X 0,Y 488.66,Z 760.612,A -85,B 0,C 180,E1 -6413.747,E2 -6413.747} C_VEL
LIN {X 0,Y 488.693,Z 760.61,A -85,B 0,C 180,E1 -6416.923,E2 -6416.923} C_VEL
LIN {X 0,Y 488.714,Z 760.608,A -85,B 0,C 180,E1 -6420.22,E2 -6420.22} C_VEL
LIN {X 0,Y 488.721,Z 760.604,A -85,B 0,C 180,E1 -6423.484,E2 -6423.484} C_VEL
LIN {X 0,Y 488.675,Z 760.614,A -85,B 0,C 180,E1 -6426.355,E2 -6426.355} C_VEL
LIN {X 0,Y 488.694,Z 760.609,A -85,B 0,C 180,E1 -6429.255,E2 -6429.255} C_VEL
LIN {X 0,Y 488.7,Z 760.607,A -85,B 0,C 180,E1 -6431.601,E2 -6431.601} C_VEL
LIN {X 0,Y 488.696,Z 760.614,A -85,B 0,C 180,E1 -6434.804,E2 -6434.804} C_VEL
LIN {X 0,Y 488.687,Z 760.609,A -85,B 0,C 180,E1 -6437.475,E2 -6437.475} C_VEL
LIN {X 0,Y 488.729,Z 760.604,A -85,B 0,C 180,E1 -6439.678,E2 -6439.678} C_VEL
LIN {X 0,Y 488.673,Z 760.615,A -85,B 0,C 180,E1 -6442.842,E2 -6442.842} C_VEL
LIN {X 0,Y 488.548,Z 760.632,A -85,B 0,C 180,E1 -6445.874,E2 -6445.874} C_VEL
LIN {X 0,Y 488.237,Z 760.671,A -85,B 0,C 180,E1 -6448.789,E2 -6448.789} C_VEL
LIN {X 0,Y 488.087,Z 760.691,A -85,B 0,C 180,E1 -6449.763,E2 -6449.763} C_VEL
LIN {X 0,Y 488.13,Z 764.759,A -85,B 0,C 180,E1 -6453.493,E2 -6453.493} C_VEL
LIN {X 0,Y 488.021,Z 767.782,A -85,B 0,C 180,E1 -6456.221,E2 -6456.221} C_VEL
LIN {X 0,Y 488.027,Z 771.243,A -85,B 0,C 180,E1 -6459.4,E2 -6459.4} C_VEL
LIN {X 0,Y 487.937,Z 774.536,A -85,B 0,C 180,E1 -6462.395,E2 -6462.395} C_VEL
LIN {X 0,Y 487.931,Z 777.806,A -85,B 0,C 180,E1 -6465.401,E2 -6465.401} C_VEL
LIN {X 0,Y 490.385,Z 790.502,A -85,B 0,C 180,E1 -6465.847,E2 -6465.847} C_VEL
LIN {X 0,Y 490.709,Z 795.999,A -85,B 0,C 180,E1 -6466.068,E2 -6466.068} C_VEL
LIN {X 0,Y 490.317,Z 807.966,A -85,B 0,C 180,E1 -6466.637,E2 -6466.637} C_VEL
LIN {X 0,Y 489.95,Z 819.35,A -85,B 0,C 180,E1 -6467.345,E2 -6467.345} C_VEL
LIN {X 0,Y 489.6,Z 830.177,A -85,B 0,C 180,E1 -6468.198,E2 -6468.198} C_VEL
LIN {X 0,Y 489.116,Z 840.692,A -85,B 0,C 180,E1 -6469.235,E2 -6469.235} C_VEL
LIN {X 0,Y 488.858,Z 849.262,A -85,B 0,C 180,E1 -6470.276,E2 -6470.276} C_VEL
LIN {X 0,Y 488.495,Z 857.632,A -85,B 0,C 180,E1 -6471.521,E2 -6471.521} C_VEL
LIN {X 0,Y 488.239,Z 865.289,A -85,B 0,C 180,E1 -6472.973,E2 -6472.973} C_VEL
LIN {X 0,Y 488.148,Z 870.41,A -85,B 0,C 180,E1 -6474.217,E2 -6474.217} C_VEL
LIN {X 0,Y 488.002,Z 874.376,A -85,B 0,C 180,E1 -6475.458,E2 -6475.458} C_VEL
LIN {X 0,Y 487.968,Z 877.308,A -85,B 0,C 180,E1 -6476.698,E2 -6476.698} C_VEL
LIN {X 0,Y 487.917,Z 878.748,A -85,B 0,C 180,E1 -6477.524,E2 -6477.524} C_VEL
LIN {X 0,Y 487.834,Z 880.37,A -85,B 0,C 180,E1 -6479.175,E2 -6479.175} C_VEL
LIN {X 0,Y 487.819,Z 880.613,A -85,B 0,C 180,E1 -6480.001,E2 -6480.001} C_VEL
LIN {X 0,Y 487.889,Z 879.848,A -85,B 0,C 180,E1 -6481.652,E2 -6481.652} C_VEL
LIN {X 0,Y 487.917,Z 878.903,A -85,B 0,C 180,E1 -6482.477,E2 -6482.477} C_VEL
LIN {X 0,Y 487.969,Z 877.527,A -85,B 0,C 180,E1 -6483.303,E2 -6483.303} C_VEL
LIN {X 0,Y 488.002,Z 874.684,A -85,B 0,C 180,E1 -6484.544,E2 -6484.544} C_VEL
LIN {X 0,Y 488.142,Z 870.817,A -85,B 0,C 180,E1 -6485.785,E2 -6485.785} C_VEL
LIN {X 0,Y 488.24,Z 865.805,A -85,B 0,C 180,E1 -6487.029,E2 -6487.029} C_VEL
LIN {X 0,Y 488.445,Z 859.458,A -85,B 0,C 180,E1 -6488.274,E2 -6488.274} C_VEL
LIN {X 0,Y 488.738,Z 851.566,A -85,B 0,C 180,E1 -6489.519,E2 -6489.519} C_VEL
LIN {X 0,Y 489.042,Z 843.495,A -85,B 0,C 180,E1 -6490.559,E2 -6490.559} C_VEL
LIN {X 0,Y 489.52,Z 833.564,A -85,B 0,C 180,E1 -6491.596,E2 -6491.596} C_VEL
LIN {X 0,Y 489.863,Z 823.781,A -85,B 0,C 180,E1 -6492.428,E2 -6492.428} C_VEL
LIN {X 0,Y 490.223,Z 813.092,A -85,B 0,C 180,E1 -6493.163,E2 -6493.163} C_VEL
LIN {X 0,Y 490.608,Z 800.518,A -85,B 0,C 180,E1 -6493.831,E2 -6493.831} C_VEL
LIN {X 0,Y 490.702,Z 792.907,A -85,B 0,C 180,E1 -6494.146,E2 -6494.146} C_VEL
LIN {X 0,Y 488.767,Z 781.706,A -85,B 0,C 180,E1 -6494.562,E2 -6494.562} C_VEL
LIN {X 0,Y 487.977,Z 778.437,A -85,B 0,C 180,E1 -6494.679,E2 -6494.679} C_VEL
LIN {X 0,Y 488.011,Z 774.739,A -85,B 0,C 180,E1 -6498.105,E2 -6498.105} C_VEL
LIN {X 0,Y 488.01,Z 771.43,A -85,B 0,C 180,E1 -6501.103,E2 -6501.103} C_VEL
LIN {X 0,Y 488.049,Z 768.415,A -85,B 0,C 180,E1 -6503.779,E2 -6503.779} C_VEL
LIN {X 0,Y 488.096,Z 764.882,A -85,B 0,C 180,E1 -6506.782,E2 -6506.782} C_VEL
LIN {X 0,Y 488.053,Z 761.563,A -85,B 0,C 180,E1 -6509.315,E2 -6509.315} C_VEL
LIN {X 0,Y 488.087,Z 760.691,A -85,B 0,C 180,E1 -6510.264,E2 -6510.264} C_VEL
LIN {X 0,Y 488.45,Z 760.646,A -85,B 0,C 180,E1 -6513.146,E2 -6513.146} C_VEL
LIN {X 0,Y 488.625,Z 760.623,A -85,B 0,C 180,E1 -6515.123,E2 -6515.123} C_VEL
LIN {X 0,Y 488.682,Z 760.61,A -85,B 0,C 180,E1 -6518.201,E2 -6518.201} C_VEL
LIN {X 0,Y 488.723,Z 760.606,A -85,B 0,C 180,E1 -6520.345,E2 -6520.345} C_VEL
LIN {X 0,Y 488.685,Z 760.611,A -85,B 0,C 180,E1 -6523.655,E2 -6523.655} C_VEL
LIN {X 0,Y 488.691,Z 760.61,A -85,B 0,C 180,E1 -6526.346,E2 -6526.346} C_VEL
LIN {X 0,Y 488.738,Z 760.608,A -85,B 0,C 180,E1 -6529.677,E2 -6529.677} C_VEL
LIN {X 0,Y 488.736,Z 760.642,A -85,B 0,C 180,E1 -6530.081,E2 -6530.081} C_VEL
LIN {X 0,Y 489.94,Z 767.406,A -85,B 0,C 180,E1 -6532.952,E2 -6532.952} C_VEL
LIN {X 0,Y 490.315,Z 771.991,A -85,B 0,C 180,E1 -6534.788,E2 -6534.788} C_VEL
LIN {X 0,Y 489.894,Z 780.35,A -85,B 0,C 180,E1 -6537.94,E2 -6537.94} C_VEL
LIN {X 0,Y 489.498,Z 789.184,A -85,B 0,C 180,E1 -6541.142,E2 -6541.142} C_VEL
LIN {X 0,Y 489.2,Z 797.382,A -85,B 0,C 180,E1 -6544.013,E2 -6544.013} C_VEL
LIN {X 0,Y 488.907,Z 806.664,A -85,B 0,C 180,E1 -6547.162,E2 -6547.162} C_VEL
LIN {X 0,Y 488.63,Z 815.999,A -85,B 0,C 180,E1 -6550.245,E2 -6550.245} C_VEL
LIN {X 0,Y 488.424,Z 825.381,A -85,B 0,C 180,E1 -6553.275,E2 -6553.275} C_VEL
LIN {X 0,Y 488.335,Z 831.69,A -85,B 0,C 180,E1 -6555.279,E2 -6555.279} C_VEL
LIN {X 0,Y 490.57,Z 845.899,A -85,B 0,C 180,E1 -6555.706,E2 -6555.706} C_VEL
LIN {X 0,Y 490.734,Z 851.528,A -85,B 0,C 180,E1 -6555.909,E2 -6555.909} C_VEL
LIN {X 0,Y 490.372,Z 863.251,A -85,B 0,C 180,E1 -6556.427,E2 -6556.427} C_VEL
LIN {X 0,Y 489.955,Z 875.243,A -85,B 0,C 180,E1 -6557.127,E2 -6557.127} C_VEL
LIN {X 0,Y 489.556,Z 886.736,A -85,B 0,C 180,E1 -6557.985,E2 -6557.985} C_VEL
LIN {X 0,Y 489.222,Z 895.752,A -85,B 0,C 180,E1 -6558.817,E2 -6558.817} C_VEL
LIN {X 0,Y 488.857,Z 905.015,A -85,B 0,C 180,E1 -6559.857,E2 -6559.857} C_VEL
LIN {X 0,Y 488.515,Z 914.036,A -85,B 0,C 180,E1 -6561.103,E2 -6561.103} C_VEL
LIN {X 0,Y 488.252,Z 921.3,A -85,B 0,C 180,E1 -6562.349,E2 -6562.349} C_VEL
LIN {X 0,Y 488.077,Z 927.666,A -85,B 0,C 180,E1 -6563.736,E2 -6563.736} C_VEL
LIN {X 0,Y 487.972,Z 932.294,A -85,B 0,C 180,E1 -6565.043,E2 -6565.043} C_VEL
LIN {X 0,Y 487.948,Z 934.61,A -85,B 0,C 180,E1 -6565.87,E2 -6565.87} C_VEL
LIN {X 0,Y 487.967,Z 936.491,A -85,B 0,C 180,E1 -6566.697,E2 -6566.697} C_VEL
LIN {X 0,Y 487.889,Z 938.899,A -85,B 0,C 180,E1 -6568.349,E2 -6568.349} C_VEL
LIN {X 0,Y 487.819,Z 939.723,A -85,B 0,C 180,E1 -6570,E2 -6570} C_VEL
LIN {X 0,Y 487.889,Z 938.893,A -85,B 0,C 180,E1 -6571.651,E2 -6571.651} C_VEL
LIN {X 0,Y 487.967,Z 936.474,A -85,B 0,C 180,E1 -6573.303,E2 -6573.303} C_VEL
LIN {X 0,Y 487.938,Z 933.497,A -85,B 0,C 180,E1 -6574.544,E2 -6574.544} C_VEL
LIN {X 0,Y 488.105,Z 929.479,A -85,B 0,C 180,E1 -6575.785,E2 -6575.785} C_VEL
LIN {X 0,Y 488.185,Z 923.278,A -85,B 0,C 180,E1 -6577.237,E2 -6577.237} C_VEL
LIN {X 0,Y 488.413,Z 916.508,A -85,B 0,C 180,E1 -6578.482,E2 -6578.482} C_VEL
LIN {X 0,Y 488.712,Z 908.098,A -85,B 0,C 180,E1 -6579.728,E2 -6579.728} C_VEL
LIN {X 0,Y 489.021,Z 899.462,A -85,B 0,C 180,E1 -6580.768,E2 -6580.768} C_VEL
LIN {X 0,Y 489.466,Z 888.812,A -85,B 0,C 180,E1 -6581.807,E2 -6581.807} C_VEL
LIN {X 0,Y 489.784,Z 878.22,A -85,B 0,C 180,E1 -6582.643,E2 -6582.643} C_VEL
LIN {X 0,Y 490.195,Z 866.716,A -85,B 0,C 180,E1 -6583.367,E2 -6583.367} C_VEL
LIN {X 0,Y 490.63,Z 853.507,A -85,B 0,C 180,E1 -6583.988,E2 -6583.988} C_VEL
LIN {X 0,Y 490.549,Z 846.041,A -85,B 0,C 180,E1 -6584.269,E2 -6584.269} C_VEL
LIN {X 0,Y 488.39,Z 832.442,A -85,B 0,C 180,E1 -6584.682,E2 -6584.682} C_VEL
LIN {X 0,Y 488.302,Z 831.078,A -85,B 0,C 180,E1 -6584.748,E2 -6584.748} C_VEL
LIN {X 0,Y 488.481,Z 820.798,A -85,B 0,C 180,E1 -6587.937,E2 -6587.937} C_VEL
LIN {X 0,Y 488.648,Z 810.777,A -85,B 0,C 180,E1 -6591.074,E2 -6591.074} C_VEL
LIN {X 0,Y 488.834,Z 802.495,A -85,B 0,C 180,E1 -6593.738,E2 -6593.738} C_VEL
LIN {X 0,Y 489.038,Z 794.362,A -85,B 0,C 180,E1 -6596.456,E2 -6596.456} C_VEL
LIN {X 0,Y 489.278,Z 786.463,A -85,B 0,C 180,E1 -6599.234,E2 -6599.234} C_VEL
LIN {X 0,Y 489.679,Z 778.791,A -85,B 0,C 180,E1 -6602.136,E2 -6602.136} C_VEL
LIN {X 0,Y 490.159,Z 772.019,A -85,B 0,C 180,E1 -6604.997,E2 -6604.997} C_VEL
LIN {X 0,Y 490.1,Z 768.765,A -85,B 0,C 180,E1 -6606.578,E2 -6606.578} C_VEL
LIN {X 0,Y 489.377,Z 764.426,A -85,B 0,C 180,E1 -6609.149,E2 -6609.149} C_VEL
LIN {X 0,Y 488.863,Z 761.32,A -85,B 0,C 180,E1 -6611.62,E2 -6611.62} C_VEL
LIN {X 0,Y 488.715,Z 760.612,A -85,B 0,C 180,E1 -6612.826,E2 -6612.826} C_VEL
LIN {X 0,Y 488.701,Z 760.613,A -85,B 0,C 180,E1 -6615.976,E2 -6615.976} C_VEL
LIN {X 0,Y 488.696,Z 760.614,A -85,B 0,C 180,E1 -6618.583,E2 -6618.583} C_VEL
LIN {X 0,Y 488.706,Z 760.613,A -85,B 0,C 180,E1 -6620.947,E2 -6620.947} C_VEL
LIN {X 0,Y 488.658,Z 760.619,A -85,B 0,C 180,E1 -6623.866,E2 -6623.866} C_VEL
LIN {X 0,Y 488.685,Z 762.15,A -85,B 0,C 180,E1 -6626.525,E2 -6626.525} C_VEL
LIN {X 0,Y 488.493,Z 764.491,A -85,B 0,C 180,E1 -6629.681,E2 -6629.681} C_VEL
LIN {X 0,Y 488.326,Z 766.838,A -85,B 0,C 180,E1 -6632.577,E2 -6632.577} C_VEL
LIN {X 0,Y 488.263,Z 769.183,A -85,B 0,C 180,E1 -6635.327,E2 -6635.327} C_VEL
LIN {X 0,Y 488.179,Z 771.588,A -85,B 0,C 180,E1 -6638.018,E2 -6638.018} C_VEL
LIN {X 0,Y 488.069,Z 774.052,A -85,B 0,C 180,E1 -6640.658,E2 -6640.658} C_VEL
LIN {X 0,Y 487.998,Z 776.53,A -85,B 0,C 180,E1 -6643.259,E2 -6643.259} C_VEL
LIN {X 0,Y 488.016,Z 778.728,A -85,B 0,C 180,E1 -6645.422,E2 -6645.422} C_VEL
LIN {X 0,Y 490.12,Z 788.831,A -85,B 0,C 180,E1 -6645.771,E2 -6645.771} C_VEL
LIN {X 0,Y 490.764,Z 794.927,A -85,B 0,C 180,E1 -6646.015,E2 -6646.015} C_VEL
LIN {X 0,Y 490.447,Z 806.287,A -85,B 0,C 180,E1 -6646.534,E2 -6646.534} C_VEL
LIN {X 0,Y 490.066,Z 818.749,A -85,B 0,C 180,E1 -6647.286,E2 -6647.286} C_VEL
LIN {X 0,Y 489.703,Z 829.215,A -85,B 0,C 180,E1 -6648.093,E2 -6648.093} C_VEL
LIN {X 0,Y 489.266,Z 838.998,A -85,B 0,C 180,E1 -6649.027,E2 -6649.027} C_VEL
LIN {X 0,Y 488.921,Z 847.883,A -85,B 0,C 180,E1 -6650.066,E2 -6650.066} C_VEL
LIN {X 0,Y 488.559,Z 856.548,A -85,B 0,C 180,E1 -6651.312,E2 -6651.312} C_VEL
LIN {X 0,Y 488.292,Z 863.444,A -85,B 0,C 180,E1 -6652.556,E2 -6652.556} C_VEL
LIN {X 0,Y 488.179,Z 869.503,A -85,B 0,C 180,E1 -6653.946,E2 -6653.946} C_VEL
LIN {X 0,Y 488.004,Z 874.487,A -85,B 0,C 180,E1 -6655.456,E2 -6655.456} C_VEL
LIN {X 0,Y 487.969,Z 877.398,A -85,B 0,C 180,E1 -6656.697,E2 -6656.697} C_VEL
LIN {X 0,Y 487.918,Z 878.801,A -85,B 0,C 180,E1 -6657.523,E2 -6657.523} C_VEL
LIN {X 0,Y 487.834,Z 880.405,A -85,B 0,C 180,E1 -6659.174,E2 -6659.174} C_VEL
LIN {X 0,Y 487.819,Z 880.634,A -85,B 0,C 180,E1 -6659.999,E2 -6659.999} C_VEL
LIN {X 0,Y 487.834,Z 880.444,A -85,B 0,C 180,E1 -6660.825,E2 -6660.825} C_VEL
LIN {X 0,Y 487.917,Z 878.887,A -85,B 0,C 180,E1 -6662.476,E2 -6662.476} C_VEL
LIN {X 0,Y 487.968,Z 877.523,A -85,B 0,C 180,E1 -6663.302,E2 -6663.302} C_VEL
LIN {X 0,Y 487.984,Z 874.657,A -85,B 0,C 180,E1 -6664.542,E2 -6664.542} C_VEL
LIN {X 0,Y 488.137,Z 870.761,A -85,B 0,C 180,E1 -6665.783,E2 -6665.783} C_VEL
LIN {X 0,Y 488.231,Z 865.738,A -85,B 0,C 180,E1 -6667.027,E2 -6667.027} C_VEL
LIN {X 0,Y 488.446,Z 859.401,A -85,B 0,C 180,E1 -6668.272,E2 -6668.272} C_VEL
LIN {X 0,Y 488.749,Z 851.471,A -85,B 0,C 180,E1 -6669.518,E2 -6669.518} C_VEL
LIN {X 0,Y 489.038,Z 843.378,A -85,B 0,C 180,E1 -6670.557,E2 -6670.557} C_VEL
LIN {X 0,Y 489.506,Z 833.493,A -85,B 0,C 180,E1 -6671.595,E2 -6671.595} C_VEL
LIN {X 0,Y 489.869,Z 822.29,A -85,B 0,C 180,E1 -6672.536,E2 -6672.536} C_VEL
LIN {X 0,Y 490.238,Z 811.435,A -85,B 0,C 180,E1 -6673.259,E2 -6673.259} C_VEL
LIN {X 0,Y 490.63,Z 799.412,A -85,B 0,C 180,E1 -6673.882,E2 -6673.882} C_VEL
LIN {X 0,Y 490.586,Z 791.991,A -85,B 0,C 180,E1 -6674.187,E2 -6674.187} C_VEL
LIN {X 0,Y 488.448,Z 780.311,A -85,B 0,C 180,E1 -6674.611,E2 -6674.611} C_VEL
